      JU    BYT0;	//-> 0 Bytes (keine)
      JU    BYT1;	//-> 1 Bytes (byte)
      JU    BYT2;	//-> 2 Bytes (word)
      JU    BYT0;	//-> 3 Bytes 
      JU    BYT4;	//-> 4 Bytes (dword)
BYT0: L     DW#16#0;	//ungueltig bzw. 0/3 Fehlerbytes
      JU    KLGO;
BYT1: L     DIB [AR1,P#0.0];	//1 Fehlerbytes
      SLD   24;	//ausrichten
      JU    KLGO;
BYT2: L     DIW [AR1,P#0.0];	//2 Fehlerbytes
      SLD   16;	//ausrichten
      JU    KLGO;
BYT4: L     DID [AR1,P#0.0];	//4 Fehlerbytes
KLGO: T     DID [AR2,P#12.0];	//in akt. Fach eintragen
      CAD;	//Tausche Akku-Inhalte (LL,LH,HL,HH)
      T     #TEMP_VAR_1;	//-> sichern
//Ermittlung der Bits in der Fehlerinfo -> Bildung eindeutiger Error-Code
      L     0;	//Bit_Zaehler initialisieren
      T     #TEMP_VAR_2;
      L     32;	//Anzahl der Bits im Dword
NXB4: T     #LOOP_CNT_1;	//-> Schleifenzaehler
      L     #TEMP_VAR_2;
      INC   1;	//Bit_Zaehler erhoehen
      T     #TEMP_VAR_2;
      L     #TEMP_VAR_1;	//Unterstes Bit rausschieben
      SRD   1;
      T     #TEMP_VAR_1;	//Wenn Fehlerbit gesetzt
      JN    ERRB;	//-> Error_Code generieren
      L     #LOOP_CNT_1;
      LOOP  NXB4;
ERRB: L     #ERROR_TYPE;	//Kanaltyp ausmaskieren
      AW    W#16#F;
      SLW   5;	//* 32 (da 32 Fehlerbits pro Kanaltyp)
      +     32;	//+ 32 (Offset)
      L     #TEMP_VAR_2;	//+ Bit_Zaehler
      +I;	//= Error_Code
      T     DIW [AR2,P#20.0];	//in akt. Fach eintragen 
      L     DIB 49;	//Fehlernummer inkrementieren
      INC   1;
      T     DIB 49;
      T     DIB [AR2,P#4.0];	//und in akt. Fach eintragen
      L     DIB 48;	//Bis vorletzter Eintrag
      L     0;
      >I;
      JC    OUT;	//-> sofort Datenausgabe
      L     P##DIAG_DAT_NORM;	//Startadresse Diagnosefach
      L     DIB 45;	//+ aktuelle Gesamtdiagnoselaenge
      SLD   3;
      +D;
      T     DID 38;	//-> neuer Error_Tippindex
      L     P##DIAG_DAT_NORM;	//Gesamtlaenge der Diagnose 
      L     DIB 44;
      SLD   3;
      +D;
      L     DID 38;	//> Error_Tippindex
      >D;
      JC    OUT;	//-> Datenausgabe 
      JU    DEND;	//sonst Diagnoseende erreicht
//Wenn kein Modulstatus oder Diagnosealarm (DS0/1) vorliegt, erfolgt 
//keine detaillierte Auswertung -> herstellerspezifische Geraetediagnose.
//Handelt es sich bei dem S7-Diagnosealarm um einen gehenden Alarm bzw.   
//sind in den S7-Alarminfos (DS0/1) keine Infos enthalten, so wird eine 
//anfaenglich uebersprungene Kennungsdiagnose anschliessend ausgewertet.
KAUS: L     DW#16#0;	//Initialisieren: Steckplatznummer,
      T     DID [AR2,P#8.0];	//Modulstatus, Kanalnummer, Kanaltyp
      T     DID [AR2,P#12.0];	//Kanal-Fehlerinfos_1
      T     DID [AR2,P#16.0];	//Kanal-Fehlerinfos_2
      T     DIW [AR2,P#20.0];	//Error-Code
      T     DIW [AR2,P#4.0];	//Error-Nr. und Error-Typ
      A     DIX 31.3;	//Wenn keine Diagnoseinfos vorliegen
      JC    NODG;	//-> allg. Geraetediagnose ausgeben
      A     DIX 31.1;	//Wenn S7-Diagnosealarm (gehend)
      A     DIX 30.7;	//und Kennungsdiagnose vorhanden
      JC    BEND;	//-> Kennungsdiagnose auswerten
      AN    DIX [AR2,P#1.0];	//Wenn Slave nicht ausgefallen
      AN    DIX [AR2,P#1.1];	//und Slave nicht gestoert
      O     DIX 31.1;	//oder S7-Diagnosealarm
      JC    NGER;	//-> keine Geraetediagnose eintragen
NODG: L     B#16#5;	//sonst Error_Typ =5 (Geraetediagnose) 
      T     #SUM_SLAVES_DIAG;	//in akt. Fach eintragen
      L     545;	//Error_Code =545
      T     DIW [AR2,P#20.0];	//in akt. Fach eintragen
//DS0 oder falscher Kanaltyp im DS1 bzw. kein Kanalfehler vorhanden
//oder allgemeine Geraetediagnose ohne Detailinfos
NCHL: L     DIB 49;	//Fehlernummer erhoehen
      INC   1;
      T     DIB 49;
      T     DIB [AR2,P#4.0];	//und in akt. Fach eintragen
NGER: L     DID 38;	//Error_Tippindex inkrementieren
      L     DIB 46;	//um die Laenge des Diagnoseblocks
      SLD   3;
      +D;
      T     DID 38;
      L     P##DIAG_DAT_NORM;	//Gesamtlaenge der Diagnose 
      L     DIB 44;
      SLD   3;
      +D;
      L     DID 38;	//> Error_Tippindex
      >D;
      JC    OUT;	//-> Datenausgabe 
      JU    DEND;	//sonst Diagnoseende erreicht
//Beginn Auswertung Modulstatus
MLGO: A     DIX 30.1;	//Wenn erstmalige Blockauswertung
      JC    MODL;
      S     DIX 30.1;	//-> Start Diagnoseblock setzen
      L     DIB 46;	//Laenge des akt. Diagnoseblocks
      DEC   4;	//- 4 Byte Headerlaenge
      SLW   2;	//* 4 Module pro Byte (2 Bits pro Modul)
      T     DIB 48;	//-> Indexzaehler im Diagnoseblock
      L     DID 38;	//Error_Tippindex um Kopfbytes erhoehen
      L     P#4.0;
      +D;
      T     DID 38;
      L     DW#16#0;	//Initialisieren: Modulnummer,
      T     DID [AR2,P#8.0];	//Modulstatus, Kanalnummer, Kanaltyp
      T     DID [AR2,P#12.0];	//Kanal-Fehlerinfos_1 
      T     DID [AR2,P#16.0];	//Kanal-Fehlerinfos_2 
      T     DIW [AR2,P#20.0];	//Error-Code
MODL: L     DIB 48;	//Indexzaehler im Diagnoseblock
LPMD: T     #LOOP_CNT_1;	//-> Schleifenzaehler
      LAR1  DID 38;
      L     DIB [AR2,P#8.0];	//Modulnummer inkrementieren 
      INC   1;	//und in akt. Fach eintragen
      T     DIB [AR2,P#8.0];
      L     DIB 48;	//Indexzaehler dekrementieren
      DEC   1;
      T     DIB 48;
      L     DID 38;	//Error_Tippindex inkrementieren
      L     P#0.2;
      +D;
      T     DID 38;
      A     DIX [AR1,P#0.0];	//Wenn Statusbits <>0
      O     DIX [AR1,P#0.1];
      JC    GFMD;	//-> Fehlerauswertung
      L     #LOOP_CNT_1;
      LOOP  LPMD;	//Wenn kein Fehler gefunden
      JU    BEND;	//-> Ende Diagnoseblock
//Fehler wird gefunden im Modulstatus
GFMD: A     DIX [AR1,P#0.0];	//Modulstatus
      =     DIX [AR2,P#9.0];	//in akt. Fach eintragen
      A     DIX [AR1,P#0.1];
      =     DIX [AR2,P#9.1];
      L     B#16#2;	//Error_Typ =2 
      T     #SUM_SLAVES_DIAG;	//in akt. Fach eintragen
      L     DIB 49;	//Fehlernummer inkrementieren
      INC   1;
      T     DIB 49;
      T     DIB [AR2,P#4.0];	//und in akt. Fach eintragen
      L     DIB 48;	//Bis vorletzter Eintrag
      L     0;
      >I;
      JC    OUT;	//-> sofort Datenausgabe
      L     P##DIAG_DAT_NORM;	//Startadresse Diagnosefach
      L     DIB 45;	//+ aktuelle Gesamtdiagnoselaenge
      SLD   3;
      +D;
      T     DID 38;	//-> neuer Error_Tippindex
      L     P##DIAG_DAT_NORM;	//Gesamtlaenge der Diagnose 
      L     DIB 44;
      SLD   3;
      +D;
      L     DID 38;	//> Error_Tippindex
      >D;
      JC    OUT;	//-> Datenausgabe 
      JU    DEND;	//sonst Diagnoseende erreicht
//Beginn Auswertung Kennungsbezogene Diagnose
//Sind neben Kennungsdiagnose noch weitere Diagnosebloecke vorhanden,
//dann wird die Kennungsdiagnose nicht ausgewertet (zu wenig Infogehalt).
//Ist aber bei S7-Slaves die Geraetediagnose ohne Infos, erfolgt nach 
//anfaenglichem Ueberspringen eine neue Auswertung der Kennungsdiagnose. 
KENB: LAR2  P##ACT_DAT;	//Startadresse aktuelles Fach
      A     DIX 30.1;	//Wenn erstmalige Blockauswertung
      JC    KNGO;
      S     DIX 30.1;	//-> Start Diagnoseblock setzen
      L     DIB 46;	//Laenge des akt. Diagnoseblocks
      DEC   1;	//- 1 Byte Headerlaenge
      SLW   3;	//* 8 Bits pro Byte
      T     DIB 48;	//-> Indexzaehler im Diagnoseblock
      L     DID 38;	//Error_Tippindex um Kopfbyte erhoehen
      L     P#1.0;
      +D;
      T     DID 38;
      L     DW#16#0;	//Initialisieren: Kennungsnummer,
      T     DID [AR2,P#8.0];	//Modulstatus, Kanalnummer, Kanaltyp
      T     DID [AR2,P#12.0];	//Kanal-Fehlerinfos_1 
      T     DID [AR2,P#16.0];	//Kanal-Fehlerinfos_2 
      T     DIW [AR2,P#20.0];	//Error-Code
KNGO: L     DIB 48;	//Indexzaehler im Diagnoseblock
LPKN: T     #LOOP_CNT_1;	//-> Schleifenzaehler
      LAR1  DID 38;
      L     DIB [AR2,P#8.0];	//Kennungsnummer inkrementieren 
      INC   1;	//und in akt. Fach eintragen
      T     DIB [AR2,P#8.0];
      L     DIB 48;	//Indexzaehler dekrementieren
      DEC   1;
      T     DIB 48;
      L     DID 38;	//Error_Tippindex inkrementieren
      L     P#0.1;
      +D;
      T     DID 38;
      A     DIX [AR1,P#0.0];	//Wenn Kennung gesetzt
      JC    GFKN;	//-> Fehlerauswertung
      L     #LOOP_CNT_1;
      LOOP  LPKN;	//Wenn kein Fehler gefunden
      JU    BEND;	//-> Ende Diagnoseblock
//Fehler wird gefunden in der Kennungsdiagnose
GFKN: A     DIX 30.7;	//Wenn Kennungsdiagnose vorhanden
      AN    DIX 31.0;	//und bisher keine Kanaldiagnose 
      AN    DIX 31.2;	//und bisher keine S7-Diagnose 
      JC    KEGO;	//-> neue bzw. weitere Auswertung
      S     DIX 30.7;	//sonst Erst-Erkennung setzen
      L     DIB 44;	//Wenn SFC13-Diagnoselaenge
      L     DIB 45;	//> aktuelle Gesamtdiagnoselaenge
      >I;
      JC    BEND;	//-> Keine Kennungsdiagnose auswerten
KEGO: L     B#16#1;	//Error_Typ =1 
      T     #SUM_SLAVES_DIAG;	//in akt. Fach eintragen
      L     DIB 49;	//Fehlernummer inkrementieren
      INC   1;
      T     DIB 49;
      T     DIB [AR2,P#4.0];	//und in akt. Fach eintragen
      L     DIB 48;	//Bis vorletzter Eintrag
      L     0;
      >I;
      JC    OUT;	//-> sofort Datenausgabe
      L     P##DIAG_DAT_NORM;	//Startadresse Diagnosefach
      L     DIB 45;	//+ aktuelle Gesamtdiagnoselaenge
      SLD   3;
      +D;
      T     DID 38;	//-> neuer Error_Tippindex
      L     P##DIAG_DAT_NORM;	//Gesamtlaenge der Diagnose 
      L     DIB 44;
      SLD   3;
      +D;
      L     DID 38;	//> Error_Tippindex
      >D;
      JC    OUT;	//-> Datenausgabe 
      JU    DEND;	//sonst Diagnoseende erreicht
//Beginn Auswertung Kanalbezogene Diagnose (immer 3 Bytes lang)
KANB: S     DIX 31.0;	//Kanaldiagnose vorhanden
      R     DIX 30.0;	//Error_TIPP-Start ruecksetzen
      LAR2  P##ACT_DAT;	//Startadresse aktuelles Fach
      L     DW#16#0;	//Initialisieren: Kennungsnummer,
      T     DID [AR2,P#8.0];	//Modulstatus, Kanalnummer, Kanaltyp
      T     DID [AR2,P#12.0];	//Kanal-Fehlerinfos_1 
      T     DID [AR2,P#16.0];	//Kanal-Fehlerinfos_2 
      T     DIW [AR2,P#20.0];	//Error-Code
      LAR1  DID 38;	//Error_Tippindex
      L     DIB [AR1,P#0.0];	//Header(Bit7,6:HeaderCode/5-0:KennungsNr)
      AW    W#16#3F;	//Kanalkennungsnummer ermitteln
      INC   1;
      T     DIB [AR2,P#8.0];	//in akt. Fach eintragen
      L     DIB [AR1,P#1.0];	//Kanalnummer ermitteln
      AW    W#16#3F;
      T     #ERROR_NO;	//in akt. Fach eintragen
      L     DIB [AR1,P#1.0];	//Kanaltyp (nach Norm) ermitteln
      SRW   6;	//00=Res, 01=In, 02=Out, 03=In/Out
      T     #ERROR_TYPE;	//in akt. Fach eintragen
//Fehlerinfo bilden, indem der ermittelte Error_Code ueber "2^Error_Code"
//bitcodiert wird.
      L     DW#16#1;	//Fehlerinfo vorbelegen
      T     #TEMP_VAR_1;
      L     B#16#0;
      L     DIB [AR1,P#2.0];	//Fehlertyp
      AW    W#16#1F;	//ausmaskieren -> Error_Code
      T     DIW [AR2,P#20.0];	//in akt. Fach eintragen
      ==I;	//Wenn Error_Code =0
      JC    NCOD;	//-> keine weitere Fehlerinfo-Kodierung 
ZEXP: T     #LOOP_CNT_1;	//Schleifenzaehler =Error_Code
      L     #TEMP_VAR_1;	//Fehlerinfo * 2 (potenzieren)
      SLD   1;
      T     #TEMP_VAR_1;
      L     #LOOP_CNT_1;
      LOOP  ZEXP;
NCOD: L     #TEMP_VAR_1;	//Bitcodierte Fehlerinfo
      CAD;	//Tausche Akku-Inhalte (LL,LH,HL,HH)   
      T     DID [AR2,P#12.0];	//in akt. Fach eintragen
      L     B#16#3;	//Error_Typ =3 
      T     #SUM_SLAVES_DIAG;	//in akt. Fach eintragen
      L     DIB 49;	//Fehlernummer inkrementieren
      INC   1;
      T     DIB 49;
      T     DIB [AR2,P#4.0];	//und in akt. Fach eintragen
      L     DID 38;	//Error_Tippindex inkrementieren
      L     P#3.0;	//um die Laenge des Diagnoseblocks
      +D;
      T     DID 38;
      L     P##DIAG_DAT_NORM;	//Gesamtlaenge der Diagnose 
      L     DIB 44;
      SLD   3;
      +D;
      L     DID 38;	//> Error_Tippindex
      >D;
      JC    OUT;	//-> Datenausgabe 
//An diese Stelle kommt das Programm nur, wenn bei der Fehlersuche im 
//Diagnoseblock ein Fehler gefunden wurde und der Error-Tippindex das 
//Ende des Diagnosetelegramms erreicht hat. Dann wird beim naechsten
//Fehler-Tippen wieder beim ersten Diagnoseblock des Diagnosetelegramms
//begonnen.
DEND: R     DIX 30.0;	//Error_TIPP-Start ruecksetzen
      L     DIB 49;	//Fehlernummer
      T     DIB [AR2,P#4.0];	//in akt. Fach eintragen
      L     6;	//Akt. Diaglaenge initialisieren
      T     DIB 45;	//mit 6 Bytes Normdiagnose
      L     0;	//Initialisieren
      T     DIB 46;	//Initialsieren Blocklaenge
      T     DIB 49;	//Fehlernummer =0 setzen
      L     P##DIAG_DAT_NORM;
      T     DID 38;	//Error_Tippindex 
      JU    OUT;	//-> Datenausgabe
//An diese Stelle kommt das Programm nur, wenn bei der Fehlersuche im 
//Diagnoseblock kein Fehler gefunden wurde. Dann wird geprueft, ob das
//Blockende auch gleichzeitig das Ende des gesamten Diagnosetelegramms
//bedeutet. Wenn ja, faengt die Fehlerauswertung sofort beim ersten 
//Diagnoseblock des Diagnosetelegramms wieder an. Ansonsten wird beim 
//naechst folgenden Diagnoseblock weiter nach Fehlern gesucht.
BEND: L     DIB 44;	//Wenn SFC13-Diagnoselaenge 
      L     DIB 45;	//> Aktuelle Gesamtdiagnoselaenge
      >I;
      JC    NBLK;	//-> naechsten Diagblock auswerten
      L     6;	//Akt. Diaglaenge initialisieren
      T     DIB 45;	//mit 6 Bytes Normdiagnose
      L     0;
      T     DIB 46;	//Initialisieren Blocklaenge
      T     DIB 49;	//Fehlernummer =0 setzen
      T     DIB 48;	//Indexzaehler im Diagblock loeschen
      T     DIB [AR2,P#8.0];	//Kennungs- bzw. Modul-Nr. loeschen 
      L     P##DIAG_DAT_NORM;
      T     DID 38;	//Error_Tippindex =Start Diagnose
      A(;
      L     DIB [AR2,P#4.0];	//Wenn bisher keine Fehler gefunden
      L     0;
      ==I;
      );
      AN    DIX 30.7;	//und keine Kenn.diagnose vorhanden
      R     DIX 30.0;	//-> Error_TIPP-Start ruecksetzen
      JC    OUT;	//-> weiter Datenausgabe
      JU    NBLK;	//sonst ersten Diagblock auswerten
NETWORK
TITLE = Versorgung der Ausgangsparameter
//Die Daten aus dem aktuellen Fach und die Anzahl der betroffenen Slaves werden 
//an die FB-Ausgangsparameter uebergeben. Zusaetzlich wird auf den Diagnose- 
//Zaehler des aktuell angezeigten Slaves zugegriffen und am Ausgangsparameter 
//angezeigt. 
OUT:  LAR2  P##ACT_DAT;	//Startadresse aktuelles Fach
      L     B#16#0;	//Wenn Slave_Nr. =0
      T     DIB 26;	//-> Diagnose_Zaehler vorab loeschen
      L     DIB [AR2,P#0.0];	//-> kein Diagnose_Zaehler auswerten 
      T     DIB 6;	//Slave_Nr. ausgeben
      ==I;
      JC    STAT;
      DEC   1;	//Slaveposition = Slave_Nr.-1
      SLD   3;	//Byteadresse
      L     P##DIAG_CNT;	//+ Startadresse Diagnose_Zaehler
      +D;
      LAR1;
      L     DIB [AR1,P#0.0];	//Diag_Zaehler des Slaves lesen
      T     DIB 26;	//und ausgeben
STAT: L     DIB [AR2,P#1.0];
      T     DIB 7;	//Slave_Status ausgeben
      L     DIW [AR2,P#2.0];
      T     DIW 8;	//Ident_Number (PNO-ID) ausgeben
      L     DIB [AR2,P#4.0];
      T     DIB 10;	//Error_Nr. ausgeben
      L     #SUM_SLAVES_DIAG;
      T     DIB 11;	//Error_Typ ausgeben
//In Fach 6 und 7 liegt die Diagnoseadresse des Slaves.
      L     DIB [AR2,P#8.0];
      T     DIB 12;	//Modul_Nr. ausgeben
      L     DIB [AR2,P#9.0];
      T     DIB 13;	//Modul_Status ausgeben
      L     #ERROR_NO;
      T     DIB 14;	//Kanal_Nr. ausgeben
      L     #ERROR_TYPE;
      T     DIB 15;	//Kanal_Typ ausgeben
      L     DIW [AR2,P#20.0];
      T     DIW 16;	//Kanal_Errorcode
      L     DID [AR2,P#12.0];
      T     DID 18;	//Kanal_Fehlerinfos_1 ausgeben
      L     DID [AR2,P#16.0];
      T     DID 22;	//Kanal_Fehlerinfos_2 ausgeben
      L     DIB 32;
      T     DIB 5;	//Summe der Betr_Slaves ausgeben
NETWORK
TITLE = OK-Bit, BUSY-Bit, Tippindex, Interrupts freigeben
//Sind keine Slaves betroffen (ausgefallen oder gestoert), wird das O.K.-Bit 
//gesetzt und der Slave- und Error-Tippindex initialisiert. Bei falscher 
//Bausteinparametrierung wird der Inhalt des Eingangsparameters Mastersystem-ID 
//in das C91-Fach eingetragen. Ist RESET aktiviert, wird die Init-Routine 
//bearbeitet. Abschliessend werden die Interrupts wieder freigegeben. 
ENDE: L     DIB 32;	//Wenn Anzahl Betr_Slaves =0
      L     0;
      ==I;
      JCN   BUSY;
      S     DIX 4.0;	//-> Alles_O.K.-Bit setzen
      R     DIX 29.7;	//-> Tippstart Slaves ruecksetzen
      R     DIX 30.0;	//-> Tippstart Fehler ruecksetzen
      L     P##AFFECT_SLAVES;	//-> Slave_Tippindex initialisieren
      T     DID 34;
      L     P##DIAG_DAT_NORM;	//-> Error_Tippindex initialisieren
      T     DID 38;
      L     1;	//-> Slaveadresse initialisieren
      T     DIW 50;
BUSY: A     DIX 1402.4;	//Wenn Reset aktiviert
      FP    DIX 29.5;
      S     DIX 30.3;	//sichern
      A     DIX 30.4;	//Wenn Parametrierfehler
      O(;	//oder
      A     DIX 28.4;	//Wenn Anlauf/Resetroutine beendet
      AN    DIX 28.7;	//     und kein SFC13-Lesen aktiv
      AN    DIX 29.0;	//     und kein SZLC91-Lesen aktiv
      A(;	//     und 
      AN    DIX 29.2;	//         kein Folgeauftrag vorh.
      O(;	//         oder
      A     DIX 29.2;	//         Folgeauftrag vorh.
      A     DIX 30.3;	//         aber Reset aktiviert  
      );
      );
      );
      R     DIX 27.1;	//-> FB-Bearbeitung beendet
      AN    DIX 30.4;	//Wenn Parametrierfehler
      JC    PROK;
      LAR1  P##SZL_READ_C91;	//Startadresse C91-Fach (BGZD)
      L     #MAST_SYSTEM_ID;	//Eingangsparameter Mastersystem-ID 
      T     DIB [AR1,P#0.0];	//in C91-Fach eintragen
PROK: AN    DIX 27.1;	//Wenn BUSY =0
      A     DIX 30.3;	//und Reset aktiv
      JC    RSET;	//-> alles initialisieren
      A     DIX 30.6;	//BIE-Bit sichern
      SAVE;
      CALL  "EN_AIRT" (
           RET_VAL                  := #RETVAL_SFC);	//Verz. Interrupts wieder freigeben
END_FUNCTION_BLOCK

// FB 523: know-how protected block, not included

// FB 913: know-how protected block, not included

// FB 914: know-how protected block, not included

// FB 915: know-how protected block, not included

FUNCTION_BLOCK "Job_List"	// FB 919
TITLE = Job_List
//V1.1
AUTHOR : SIEMENS
FAMILY : COMM
NAME : JOB_LIST
VERSION : 1.1
VAR_INPUT
  CYCLICAL : TIME ;	//Cyclical time to start the job list
  DONE : BOOL ;	//Job finished without error (from MODBUS block)
  ERROR : BOOL ;	//Job finished with error (from MODBUS block)
  Job1_DATA_TYPE : BYTE ;	//1st job: data type (1-4)
  Job1_START_ADDRESS : WORD ;	//Start address (register or bit)
  Job1_LENGTH : WORD ;	//Count of registers/bits
  Job1_WRITE_READ : BOOL ;	//TRUE = write, FALSE = read
  Job2_DATA_TYPE : BYTE ;	//2nd job: data type (1-4)
  Job2_START_ADDRESS : WORD ;	//Start address (register or bit)
  Job2_LENGTH : WORD ;	//Count of registers/bits
  Job2_WRITE_READ : BOOL ;	//TRUE = write, FALSE = read
  Job3_DATA_TYPE : BYTE ;	//3rd job: data type (1-4)
  Job3_START_ADDRESS : WORD ;	//Start address (register or bit)
  Job3_LENGTH : WORD ;	//Count of registers/bits
  Job3_WRITE_READ : BOOL ;	//TRUE = write, FALSE = read
  Job4_DATA_TYPE : BYTE ;	//4th job: data type (1-4)
  Job4_START_ADDRESS : WORD ;	//Start address (register or bit)
  Job4_LENGTH : WORD ;	//Count of registers/bits
  Job4_WRITE_READ : BOOL ;	//TRUE = write, FALSE = read
  Job5_DATA_TYPE : BYTE ;	//5th job: data type (1-4)
  Job5_START_ADDRESS : WORD ;	//Start address (register or bit)
  Job5_LENGTH : WORD ;	//Count of registers/bits
  Job5_WRITE_READ : BOOL ;	//TRUE = write, FALSE = read
  Job6_DATA_TYPE : BYTE ;	//1st job: data type (1-4)
  Job6_START_ADDRESS : WORD ;	//Start address (register or bit)
  Job6_LENGTH : WORD ;	//Count of registers/bits
  Job6_WRITE_READ : BOOL ;	//TRUE = write, FALSE = read
  Job7_DATA_TYPE : BYTE ;	//2nd job: data type (1-4)
  Job7_START_ADDRESS : WORD ;	//Start address (register or bit)
  Job7_LENGTH : WORD ;	//Count of registers/bits
  Job7_WRITE_READ : BOOL ;	//TRUE = write, FALSE = read
  Job8_DATA_TYPE : BYTE ;	//3rd job: data type (1-4)
  Job8_START_ADDRESS : WORD ;	//Start address (register or bit)
  Job8_LENGTH : WORD ;	//Count of registers/bits
  Job8_WRITE_READ : BOOL ;	//TRUE = write, FALSE = read
  Job9_DATA_TYPE : BYTE ;	//4th job: data type (1-4)
  Job9_START_ADDRESS : WORD ;	//Start address (register or bit)
  Job9_LENGTH : WORD ;	//Count of registers/bits
  Job9_WRITE_READ : BOOL ;	//TRUE = write, FALSE = read
  Job10_DATA_TYPE : BYTE ;	//5th job: data type (1-4)
  Job10_START_ADDRESS : WORD ;	//Start address (register or bit)
  Job10_LENGTH : WORD ;	//Count of registers/bits
  Job10_WRITE_READ : BOOL ;	//TRUE = write, FALSE = read
END_VAR
VAR_OUTPUT
  QENQ : BOOL ;	//Job initiation
  QDATA_TYPE : BYTE ;	//Data type 1:Coils, 2:Inputs, 3:Holding, 4:Input Registers
  QSTART_ADDRESS : WORD ;	//Start address (register or bit)
  QLENGTH : WORD ;	//Count of registers/bits
  QWRITE_READ : BOOL ;	//TRUE = write, FALSE = read
  BUSY : BOOL ;	//Job list processing
  STATUS : WORD ;	//Status information of job list block
END_VAR
VAR_IN_OUT
  ABORT : BOOL ;	//Reset: Stop the processing of the job list
END_VAR
VAR
  Count_of_Jobs : INT  := 10;	//Count of Jobs in the input area
  TON_JOB : SFB 4;	//Timer for cyclical processing
  Current_Job : INT ;	//Current processed job
  i : INT ;	//internal counter
  sIDB_Nr : WORD ;	//number of instance data block
  Next_Job : BOOL ;	//TRUE: next job should be start
  Wait : BOOL ;	//internal use
END_VAR
VAR_TEMP
  address_Struct : STRUCT
   ANY_id : WORD ;
   Length : WORD ;
   DB_Number : WORD ;
   Byte_Pointer : DWORD ;
  END_STRUCT ;
END_VAR
BEGIN
// body was compiled from an SCL source; compiled code not shown
END_FUNCTION_BLOCK

FUNCTION_BLOCK "JOB_RESET"	// FB 921
VERSION : 0.0
VAR_INPUT
  CMD : BOOL ;
  SOURSE_DB : BLOCK_DB ;
  TARGET_DB : BLOCK_DB ;
END_VAR
VAR
  I : INT ;	//Static Variables
END_VAR
BEGIN
// body was compiled from an SCL source; compiled code not shown
END_FUNCTION_BLOCK

// FB 1071: know-how protected block, not included

// FB 1501: know-how protected block, not included

FUNCTION_BLOCK "HF3_PID_FB2005"	// FB 2005
TITLE = PID
VERSION : 0.1
VAR_INPUT
  COM_RST : BOOL ;
  MAN_ON { S7_m_c := 'true' }: BOOL  := TRUE;	//1-手动，0-自动
  PVPER_ON : BOOL ;	//0-设定的过程变量；1-来自IO的过程变量
  P_SEL : BOOL  := TRUE;	//P 选择开关
  I_SEL : BOOL  := TRUE;	//I 选择开关
  INT_HOLD : BOOL ;	//INTEGRAL ACTION HOLD 积分器被冻结
  I_ITL_ON : BOOL ;	//INITIALIZATION OF THE INTEGRAL 积分器初始值
  D_SEL : BOOL ;	//DERIVATIVE ACTION ON可以单独激活或失去D作用
  INT_EXT { S7_m_c := 'true' }: BOOL ;	//0＝内部设定，1＝外部设定
  IN_1 : BOOL ;	//Spare
  IN_2 : BOOL ;	//Spare
  IN_3 : BOOL ;	//Backup
  PV_PER : WORD ;	//PROCESS VARIABLE PERIPHERAL
  SP_INT { S7_m_c := 'true'; S7_archive := 'shortterm' }: REAL ;	//PID内部设定值
  UNIT { S7_m_c := 'true' }: INT ;	//Unit
  PV_IN { S7_m_c := 'true'; S7_archive := 'shortterm' }: REAL ;	//实际输入值
  GAIN { S7_m_c := 'true' }: REAL  := 2.000000e+000;	//比例
  TI { S7_m_c := 'true' }: DINT  := L#10;	//积分时间
  TD { S7_m_c := 'true' }: DINT  := L#10;	//微分时间
  CYCLE : TIME  := T#1S;
  TM_LAG : TIME  := T#2S;	//TIME LAG OF THE DERIVATIVE ACTION微分延时时间
  DEADB_W { S7_m_c := 'true' }: REAL ;	//死区
  LMN_HLM { S7_m_c := 'true' }: REAL  := 1.000000e+002;	//输出上限
  LMN_LLM { S7_m_c := 'true' }: REAL ;	//输出下限
  PV_FAC : REAL  := 1.000000e+000;	//实际输入因子  （通常为"1"）
  PV_OFF : REAL ;	//实际输入补偿  （通常不需要）
  LMN_FAC : REAL  := 1.000000e+000;	//输出因子  （通常为"1"）
  LMN_OFF : REAL ;	//输出补偿  （通常不需要）
  I_ITLVAL : REAL ;	//积分初始值
  DISV : REAL ;	//前馈值
  SP_EXT { S7_m_c := 'true' }: REAL ;	//逻辑外部设定值（外环输出值）
  IN_4 : REAL ;	//Spare
  PV_RANG_L : REAL ;
  PV_RANG_H : REAL  := 1.000000e+002;
END_VAR
VAR_OUTPUT
  QLMN_HLM : BOOL ;	//手动值高限
  QLMN_LLM : BOOL ;	//手动值底限
  QMAN_ON { S7_m_c := 'true' }: BOOL ;	//PID手自动状态，0-手动，1-自动
  OUT_1 : BOOL ;	//Spare
  OUT_2 : BOOL ;	//Spare
  OUT_3 : BOOL ;	//Spare
  LMN_PER { S7_m_c := 'true' }: WORD ;	//预设手动值
  LMN_P { S7_m_c := 'true' }: REAL ;	//PROPORTIONAL COMPONENT
  LMN_I { S7_m_c := 'true' }: REAL ;	//INTEGRAL COMPONENT
  LMN_D { S7_m_c := 'true' }: REAL ;	//DERIVATIVE COMPONENT
  PV { S7_m_c := 'true' }: REAL ;	//过程值
  ER { S7_m_c := 'true' }: REAL ;	//错误信号
  OUT_4 : BOOL ;	//Spare
END_VAR
VAR_IN_OUT
  MAN { S7_m_c := 'true'; S7_archive := 'shortterm' }: REAL ;	//手动输出值
  LMN { S7_m_c := 'true'; S7_archive := 'shortterm' }: REAL ;	//PID输出
  IN_OUT_1 : BOOL ;
  IN_OUT_2 : BOOL ;
  IN_OUT_3 : REAL ;
  SP_M { S7_m_c := 'true' }: REAL ;	//SP实际设定值
END_VAR
VAR
  PID_CTRL : FB 41;
  TI_M : DINT ;
  TD_M : DINT ;
  TI_TIME : TIME ;
  TD_TIME : TIME ;
END_VAR
BEGIN
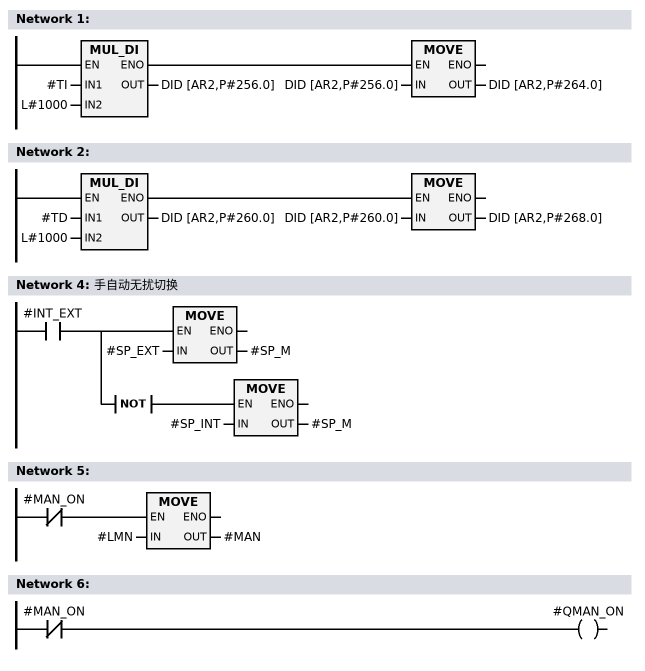
NETWORK
TITLE =
//Intergration Time
      A(;
      L     #TI;
      L     L#1000;
      *D;
      T     DID [AR2,P#256.0];
      AN    OV;
      SAVE;
      CLR;
      A     BR;
      );
      JNB   _001;
      L     DID [AR2,P#256.0];
      T     DID [AR2,P#264.0];
_001: NOP   0;
NETWORK
TITLE =
//Derivative Time
      A(;
      L     #TD;
      L     L#1000;
      *D;
      T     DID [AR2,P#260.0];
      AN    OV;
      SAVE;
      CLR;
      A     BR;
      );
      JNB   _002;
      L     DID [AR2,P#260.0];
      T     DID [AR2,P#268.0];
_002: NOP   0;
NETWORK
TITLE =
//Cont_C
      A     #COM_RST;
      =     L 0.0;
      BLD   103;
      A     #MAN_ON;
      =     L 0.1;
      BLD   103;
      A     #PVPER_ON;
      =     L 0.2;
      BLD   103;
      A     #P_SEL;
      =     L 0.3;
      BLD   103;
      A     #I_SEL;
      =     L 0.4;
      BLD   103;
      A     #INT_HOLD;
      =     L 0.5;
      BLD   103;
      A     #I_ITL_ON;
      =     L 0.6;
      BLD   103;
      A     #D_SEL;
      =     L 0.7;
      BLD   103;
      BLD   14;
      =     L 7.0;
      L     DINO;
      T     LW 5;
      CDB;
      OPN   DI [LW 5];
      TAR2  LD 1;
      A     L 0.0;
      =     DIX [AR2,P#130.0];
      A     L 0.1;
      =     DIX [AR2,P#130.1];
      A     L 0.2;
      =     DIX [AR2,P#130.2];
      A     L 0.3;
      =     DIX [AR2,P#130.3];
      A     L 0.4;
      =     DIX [AR2,P#130.4];
      A     L 0.5;
      =     DIX [AR2,P#130.5];
      A     L 0.6;
      =     DIX [AR2,P#130.6];
      A     L 0.7;
      =     DIX [AR2,P#130.7];
      L     DBD [AR2,P#26.0];
      T     DID [AR2,P#132.0];
      L     DBD [AR2,P#126.0];
      T     DID [AR2,P#136.0];
      L     DBD [AR2,P#10.0];
      T     DID [AR2,P#140.0];
      L     DBW [AR2,P#2.0];
      T     DIW [AR2,P#144.0];
      L     DBD [AR2,P#112.0];
      T     DID [AR2,P#146.0];
      L     DBD [AR2,P#14.0];
      T     DID [AR2,P#150.0];
      L     DBD [AR2,P#264.0];
      T     DID [AR2,P#154.0];
      L     DBD [AR2,P#268.0];
      T     DID [AR2,P#158.0];
      L     DBD [AR2,P#30.0];
      T     DID [AR2,P#162.0];
      L     DBD [AR2,P#34.0];
      T     DID [AR2,P#166.0];
      L     DBD [AR2,P#38.0];
      T     DID [AR2,P#170.0];
      L     DBD [AR2,P#42.0];
      T     DID [AR2,P#174.0];
      L     DBD [AR2,P#46.0];
      T     DID [AR2,P#178.0];
      L     DBD [AR2,P#50.0];
      T     DID [AR2,P#182.0];
      L     DBD [AR2,P#54.0];
      T     DID [AR2,P#186.0];
      L     DBD [AR2,P#58.0];
      T     DID [AR2,P#190.0];
      L     DBD [AR2,P#62.0];
      T     DID [AR2,P#194.0];
      L     DBD [AR2,P#66.0];
      T     DID [AR2,P#198.0];
      +AR2  P#130.0;
      UC    "pid";
      LAR2  LD 1;
      L     DID [AR2,P#202.0];
      T     DBD [AR2,P#116.0];
      L     DIW [AR2,P#206.0];
      T     DBW [AR2,P#88.0];
      A     DIX [AR2,P#208.0];
      =     DBX [AR2,P#86.0];
      A     DIX [AR2,P#208.1];
      =     DBX [AR2,P#86.1];
      L     DID [AR2,P#210.0];
      T     DBD [AR2,P#90.0];
      L     DID [AR2,P#214.0];
      T     DBD [AR2,P#94.0];
      L     DID [AR2,P#218.0];
      T     DBD [AR2,P#98.0];
      L     DID [AR2,P#222.0];
      T     DBD [AR2,P#102.0];
      L     DID [AR2,P#226.0];
      T     DBD [AR2,P#106.0];
      CDB;
      BLD   15;
      NOP   0;
NETWORK
TITLE = 手自动无扰切换
//当外部设定时，逻辑外部设定值赋值给设定值；当内部设定时，PID内部设定值赋值给设定
//值
//。
//主要用在串级调节回路
      A     #INT_EXT;
      =     L 0.0;
      A     L 0.0;
      JNB   _003;
      L     #SP_EXT;
      T     #SP_M;
_003: NOP   0;
      A     L 0.0;
      NOT;
      JNB   _004;
      L     #SP_INT;
      T     #SP_M;
_004: NOP   0;
NETWORK
TITLE =
      AN    #MAN_ON;
      JNB   _005;
      L     #LMN;
      T     #MAN;
_005: NOP   0;
NETWORK
TITLE =
      AN    #MAN_ON;
      =     #QMAN_ON;
END_FUNCTION_BLOCK

FUNCTION_BLOCK "HF3_RunFaultSum"	// FB 2006
TITLE = TIMER_MOTOR
AUTHOR : SIEMENS
FAMILY : SIEMENS
NAME : SIEMENS
VERSION : 1.0
VAR_INPUT
  RUN : BOOL ;
  ERROR : BOOL ;
  SAMPLE_T : BOOL ;	//Cycle Time of the CPU Time plus (Seconds)
  RESET_RUN : BOOL ;
  RESET_ERROR : BOOL ;
  RESET_TIME : BOOL ;
END_VAR
VAR_OUTPUT
  RUNTIME : REAL ;	//Run Timer in Hour
  RUN_COUNTER : INT ;
  ERROR_COUNTER : INT ;
END_VAR
VAR
  RUN_SECOND : REAL ;	//RUNTIME counter in Second
  OLD_SAMPLE_T : BOOL ;
  OLD_RUN : BOOL ;
  OLD_ERROR : BOOL ;
END_VAR
BEGIN
// body was compiled from an SCL source; compiled code not shown
END_FUNCTION_BLOCK

FUNCTION_BLOCK "HF3_EPS_FB2501"	// FB 2501
TITLE = EPS 主程序端
//定义参照点表
VERSION : 0.1
VAR
  EPS21 : FB 2502;
  EPS11 : FB 2502;
END_VAR
BEGIN
NETWORK
TITLE = EPS_A
// (network holds code this reader does not know; not shown)
NETWORK
TITLE =
// (network holds code this reader does not know; not shown)
END_FUNCTION_BLOCK

FUNCTION_BLOCK "HF3_EPS_FB2502"	// FB 2502
VERSION : 0.1
VAR_INPUT
  DB_Number : INT ;
END_VAR
VAR_OUTPUT
  EPS_ToHMI1 : WORD ;
  EPS_ToHMI : ARRAY  [0 .. 15 ] OF INT ;
END_VAR
VAR
  data_p : DWORD ;	//DATA POINTER
  AR2_data : DWORD ;
END_VAR
VAR_TEMP
  dbnumber : INT ;
  DIN_TEMP : WORD ;
  NO_TEMP : INT ;
  CommOK : BOOL ;	//communication status
  AR2_Temp : DWORD ;	//current multi-instance AR2 data
END_VAR
BEGIN
NETWORK
TITLE = Initialize Parameters
      L     P#2.0;
      T     #data_p;
      L     DW#16#0;
      T     #AR2_Temp;
      L     #DB_Number;
      T     #dbnumber;
      OPN   DB [#dbnumber];
      L     DINO;
      T     #DIN_TEMP;
      OPN   DI [#DIN_TEMP];
NETWORK
TITLE = Data Output
      L     #data_p;
      LAR1;
      TAR2;
//Figure out the absolute address of Instance DB variable 
      T     #AR2_Temp;
      AD    DW#16#FFFFFF;	//Close area identifier 
      L     P##EPS_ToHMI;
      +D;
      LAR2;
//  Pass PARAMETER
      L     16;
LP:   T     #NO_TEMP;
      L     DBW [AR1,P#0.0];
      T     W [AR2,P#0.0];
      +AR1  P#2.0;
      +AR2  P#2.0;
      L     #NO_TEMP;
      LOOP  LP;
      L     #AR2_Temp;	// Recovery AR2   
      LAR2;
NETWORK
TITLE = Communication Status
      L     DBW 0;
      L     0;
      ==I;
      =     #CommOK;
NETWORK
TITLE = Pass EPS Status to HMI
      CALL  "HF3_B_T_W_FC51" (
           Bit_0                    := DBX 35.0,
           Bit_1                    := DBX 35.1,
           Bit_2                    := DBX 35.2,
           Bit_3                    := DBX 35.3,
           Bit_4                    := DBX 35.4,
           Bit_5                    := DBX 35.5,
           Bit_6                    := DBX 35.6,
           Bit_7                    := DBX 35.7,
           Bit_8                    := DBX 34.0,
           Bit_9                    := DBX 34.1,
           Bit_10                   := DBX 34.2,
           Bit_11                   := DBX 34.3,
           Bit_12                   := DBX 34.4,
           Bit_13                   := DBX 34.5,
           Bit_14                   := DBX 34.6,
           Bit_15                   := #CommOK,
           Word1                    := #EPS_ToHMI1);	//市电状态(报警点) / 逆变状态(报警点) / 综合故障(报警点) / 过载(报警点) / 强制运行(报警点) / 电池状态(报警点) / 充电状态(报警点) / 支路故障(报警点) / 电池欠压 / 市电/逆变状态 / 均/浮充 / 双切位置 / ͨѶ״̬
NETWORK
TITLE = END function block
      SET;
      SAVE;
      CLR;
      BEU;
END_FUNCTION_BLOCK

FUNCTION_BLOCK "HF3_IMCC_CommOK_FB2512"	// FB 2512
VERSION : 0.1
VAR
  CommOK : FB 2513;
END_VAR
BEGIN
NETWORK
TITLE =
      BLD   14;
      =     L 6.0;
      L     DINO;
      T     LW 4;
      CDB;
      OPN   DI [LW 4];
      TAR2  LD 0;
      OPN   DI 2291;
      L     DIW 0;
      OPN   DI [LW 4];
      T     #CommOK.inRD_IMCC_HB;
      +AR2  P#0.0;
      UC    "HF3_IMCC_CommOK_FB2513";
      LAR2  LD 0;
      A     #CommOK.IMCC_CommOK;
      =     "IMCC_Comok";
      CDB;
      BLD   15;
      NOP   0;
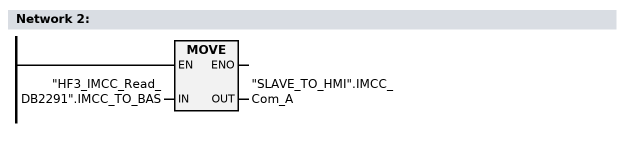
NETWORK
TITLE =
      L     "HF3_IMCC_Read_DB2291".IMCC_TO_BAS;
      T     "SLAVE_TO_HMI".IMCC_Com_A;
      NOP   0;
END_FUNCTION_BLOCK

FUNCTION_BLOCK "HF3_IMCC_CommOK_FB2513"	// FB 2513
VERSION : 0.1
VAR_INPUT
  inRD_IMCC_HB : WORD ;
END_VAR
VAR_OUTPUT
  IMCC_CommOK : BOOL ;
END_VAR
VAR
  Ton1 : SFB 4;
  CommOK1 : BOOL ;
  CommOK2 : BOOL ;
  fault1 : BOOL ;
  Ton2 : SFB 4;
  fault2 : BOOL ;
  TON3 : SFB 4;
END_VAR
BEGIN
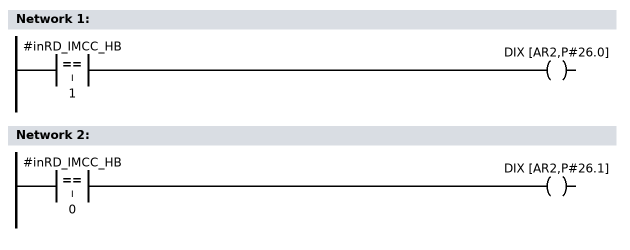
NETWORK
TITLE =
      L     #inRD_IMCC_HB;
      L     1;
      ==I;
      =     DIX [AR2,P#26.0];
NETWORK
TITLE =
      L     #inRD_IMCC_HB;
      L     0;
      ==I;
      =     DIX [AR2,P#26.1];
NETWORK
TITLE =
      A     DIX [AR2,P#26.0];
      =     L 0.0;
      BLD   103;
      BLD   16;
      =     L 7.0;
      L     DINO;
      T     LW 5;
      CDB;
      OPN   DI [LW 5];
      TAR2  LD 1;
      A     L 0.0;
      =     DIX [AR2,P#4.0];
      L     L#30000;
      T     DID [AR2,P#6.0];
      +AR2  P#4.0;
      UC    "TON";
      LAR2  LD 1;
      A     DIX [AR2,P#10.0];
      =     DBX [AR2,P#26.2];
      CDB;
      BLD   17;
      NOP   0;
NETWORK
TITLE =
      A     DIX [AR2,P#26.1];
      =     L 0.0;
      BLD   103;
      BLD   16;
      =     L 7.0;
      L     DINO;
      T     LW 5;
      CDB;
      OPN   DI [LW 5];
      TAR2  LD 1;
      A     L 0.0;
      =     DIX [AR2,P#28.0];
      L     L#30000;
      T     DID [AR2,P#30.0];
      +AR2  P#28.0;
      UC    "TON";
      LAR2  LD 1;
      A     DIX [AR2,P#34.0];
      =     DBX [AR2,P#50.0];
      CDB;
      BLD   17;
      NOP   0;
NETWORK
TITLE =
      AN    DIX [AR2,P#50.0];
      AN    DIX [AR2,P#26.2];
      =     L 0.0;
      BLD   103;
      BLD   16;
      =     L 7.0;
      L     DINO;
      T     LW 5;
      CDB;
      OPN   DI [LW 5];
      TAR2  LD 1;
      A     L 0.0;
      =     DIX [AR2,P#52.0];
      L     L#30000;
      T     DID [AR2,P#54.0];
      +AR2  P#52.0;
      UC    "TON";
      LAR2  LD 1;
      A     DIX [AR2,P#58.0];
      =     DBX [AR2,P#2.0];
      CDB;
      BLD   17;
      NOP   0;
END_FUNCTION_BLOCK

FUNCTION_BLOCK "HF3_LSQK_FB2521"	// FB 2521
VERSION : 0.1
VAR
  PT : TIME  := T#40MS;
  LSQK : FB 2522;
END_VAR
BEGIN
NETWORK
TITLE =
      BLD   14;
      =     L 7.0;
      L     DINO;
      T     LW 5;
      CDB;
      OPN   DI [LW 5];
      TAR2  LD 1;
      OPN   DI 6001;
      L     DIW 12;
      OPN   DI [LW 5];
      T     #LSQK.SCtrl;
      OPN   DI 2185;
      L     DIW 2;
      OPN   DI [LW 5];
      T     #LSQK.inRD;
      OPN   DI 2185;
      L     DIW 0;
      OPN   DI [LW 5];
      T     #LSQK.inRD_Statu;
      +AR2  P#4.0;
      UC    "HF3_LSQK_FB2522";
      LAR2  LD 1;
      L     #LSQK.qnWR;
      OPN   DI 2183;
      T     DIW 8;
      OPN   DI [LW 5];
      L     #LSQK.ToHMI;
      OPN   DI 6002;
      T     DIW 120;
      OPN   DI [LW 5];
      CDB;
      BLD   15;
      NOP   0;
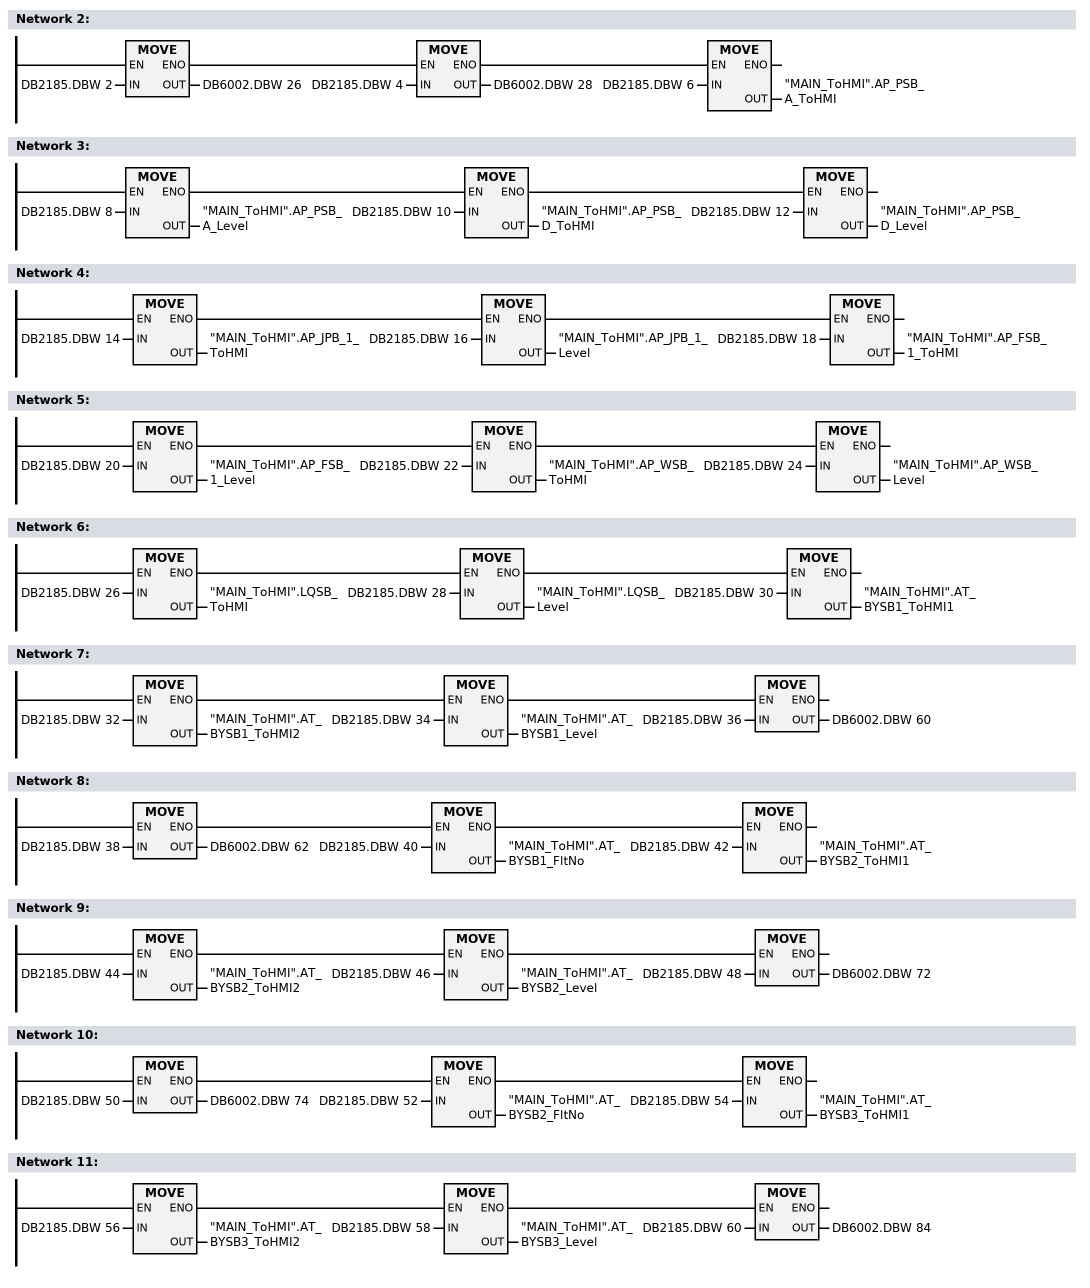
NETWORK
TITLE =
      A(;
      A(;
      L     DB2185.DBW 2;
      T     DB6002.DBW 26;
      SET;
      SAVE;
      CLR;
      A     BR;
      );
      JNB   _001;
      L     DB2185.DBW 4;
      T     DB6002.DBW 28;
      SET;
      SAVE;
      CLR;
_001: A     BR;
      );
      JNB   _002;
      L     DB2185.DBW 6;
      T     "MAIN_ToHMI".AP_PSB_A_ToHMI;
_002: NOP   0;
NETWORK
TITLE =
      A(;
      A(;
      L     DB2185.DBW 8;
      T     "MAIN_ToHMI".AP_PSB_A_Level;
      SET;
      SAVE;
      CLR;
      A     BR;
      );
      JNB   _003;
      L     DB2185.DBW 10;
      T     "MAIN_ToHMI".AP_PSB_D_ToHMI;
      SET;
      SAVE;
      CLR;
_003: A     BR;
      );
      JNB   _004;
      L     DB2185.DBW 12;
      T     "MAIN_ToHMI".AP_PSB_D_Level;
_004: NOP   0;
NETWORK
TITLE =
      A(;
      A(;
      L     DB2185.DBW 14;
      T     "MAIN_ToHMI".AP_JPB_1_ToHMI;
      SET;
      SAVE;
      CLR;
      A     BR;
      );
      JNB   _005;
      L     DB2185.DBW 16;
      T     "MAIN_ToHMI".AP_JPB_1_Level;
      SET;
      SAVE;
      CLR;
_005: A     BR;
      );
      JNB   _006;
      L     DB2185.DBW 18;
      T     "MAIN_ToHMI".AP_FSB_1_ToHMI;
_006: NOP   0;
NETWORK
TITLE =
      A(;
      A(;
      L     DB2185.DBW 20;
      T     "MAIN_ToHMI".AP_FSB_1_Level;
      SET;
      SAVE;
      CLR;
      A     BR;
      );
      JNB   _007;
      L     DB2185.DBW 22;
      T     "MAIN_ToHMI".AP_WSB_ToHMI;
      SET;
      SAVE;
      CLR;
_007: A     BR;
      );
      JNB   _008;
      L     DB2185.DBW 24;
      T     "MAIN_ToHMI".AP_WSB_Level;
_008: NOP   0;
NETWORK
TITLE =
      A(;
      A(;
      L     DB2185.DBW 26;
      T     "MAIN_ToHMI".LQSB_ToHMI;
      SET;
      SAVE;
      CLR;
      A     BR;
      );
      JNB   _009;
      L     DB2185.DBW 28;
      T     "MAIN_ToHMI".LQSB_Level;
      SET;
      SAVE;
      CLR;
_009: A     BR;
      );
      JNB   _00a;
      L     DB2185.DBW 30;
      T     "MAIN_ToHMI".AT_BYSB1_ToHMI1;
_00a: NOP   0;
NETWORK
TITLE =
      A(;
      A(;
      L     DB2185.DBW 32;
      T     "MAIN_ToHMI".AT_BYSB1_ToHMI2;
      SET;
      SAVE;
      CLR;
      A     BR;
      );
      JNB   _00b;
      L     DB2185.DBW 34;
      T     "MAIN_ToHMI".AT_BYSB1_Level;
      SET;
      SAVE;
      CLR;
_00b: A     BR;
      );
      JNB   _00c;
      L     DB2185.DBW 36;
      T     DB6002.DBW 60;
_00c: NOP   0;
NETWORK
TITLE =
      A(;
      A(;
      L     DB2185.DBW 38;
      T     DB6002.DBW 62;
      SET;
      SAVE;
      CLR;
      A     BR;
      );
      JNB   _00d;
      L     DB2185.DBW 40;
      T     "MAIN_ToHMI".AT_BYSB1_FltNo;
      SET;
      SAVE;
      CLR;
_00d: A     BR;
      );
      JNB   _00e;
      L     DB2185.DBW 42;
      T     "MAIN_ToHMI".AT_BYSB2_ToHMI1;
_00e: NOP   0;
NETWORK
TITLE =
      A(;
      A(;
      L     DB2185.DBW 44;
      T     "MAIN_ToHMI".AT_BYSB2_ToHMI2;
      SET;
      SAVE;
      CLR;
      A     BR;
      );
      JNB   _00f;
      L     DB2185.DBW 46;
      T     "MAIN_ToHMI".AT_BYSB2_Level;
      SET;
      SAVE;
      CLR;
_00f: A     BR;
      );
      JNB   _010;
      L     DB2185.DBW 48;
      T     DB6002.DBW 72;
_010: NOP   0;
NETWORK
TITLE =
      A(;
      A(;
      L     DB2185.DBW 50;
      T     DB6002.DBW 74;
      SET;
      SAVE;
      CLR;
      A     BR;
      );
      JNB   _011;
      L     DB2185.DBW 52;
      T     "MAIN_ToHMI".AT_BYSB2_FltNo;
      SET;
      SAVE;
      CLR;
_011: A     BR;
      );
      JNB   _012;
      L     DB2185.DBW 54;
      T     "MAIN_ToHMI".AT_BYSB3_ToHMI1;
_012: NOP   0;
NETWORK
TITLE =
      A(;
      A(;
      L     DB2185.DBW 56;
      T     "MAIN_ToHMI".AT_BYSB3_ToHMI2;
      SET;
      SAVE;
      CLR;
      A     BR;
      );
      JNB   _013;
      L     DB2185.DBW 58;
      T     "MAIN_ToHMI".AT_BYSB3_Level;
      SET;
      SAVE;
      CLR;
_013: A     BR;
      );
      JNB   _014;
      L     DB2185.DBW 60;
      T     DB6002.DBW 84;
_014: NOP   0;
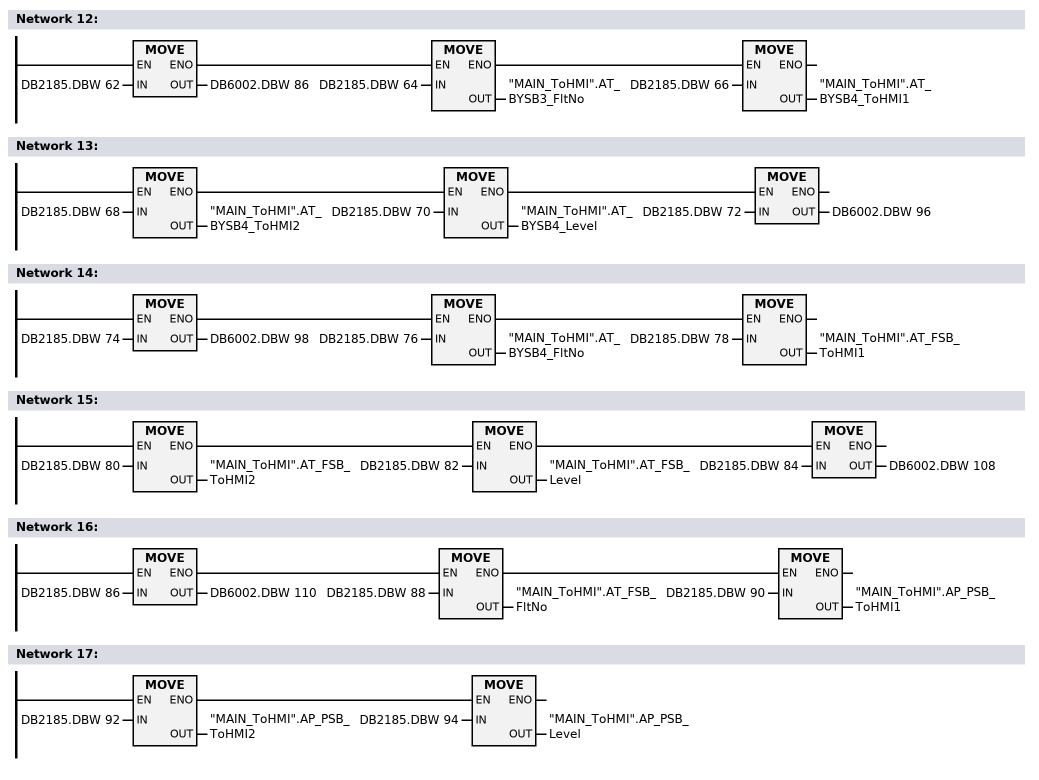
NETWORK
TITLE =
      A(;
      A(;
      L     DB2185.DBW 62;
      T     DB6002.DBW 86;
      SET;
      SAVE;
      CLR;
      A     BR;
      );
      JNB   _015;
      L     DB2185.DBW 64;
      T     "MAIN_ToHMI".AT_BYSB3_FltNo;
      SET;
      SAVE;
      CLR;
_015: A     BR;
      );
      JNB   _016;
      L     DB2185.DBW 66;
      T     "MAIN_ToHMI".AT_BYSB4_ToHMI1;
_016: NOP   0;
NETWORK
TITLE =
      A(;
      A(;
      L     DB2185.DBW 68;
      T     "MAIN_ToHMI".AT_BYSB4_ToHMI2;
      SET;
      SAVE;
      CLR;
      A     BR;
      );
      JNB   _017;
      L     DB2185.DBW 70;
      T     "MAIN_ToHMI".AT_BYSB4_Level;
      SET;
      SAVE;
      CLR;
_017: A     BR;
      );
      JNB   _018;
      L     DB2185.DBW 72;
      T     DB6002.DBW 96;
_018: NOP   0;
NETWORK
TITLE =
      A(;
      A(;
      L     DB2185.DBW 74;
      T     DB6002.DBW 98;
      SET;
      SAVE;
      CLR;
      A     BR;
      );
      JNB   _019;
      L     DB2185.DBW 76;
      T     "MAIN_ToHMI".AT_BYSB4_FltNo;
      SET;
      SAVE;
      CLR;
_019: A     BR;
      );
      JNB   _01a;
      L     DB2185.DBW 78;
      T     "MAIN_ToHMI".AT_FSB_ToHMI1;
_01a: NOP   0;
NETWORK
TITLE =
      A(;
      A(;
      L     DB2185.DBW 80;
      T     "MAIN_ToHMI".AT_FSB_ToHMI2;
      SET;
      SAVE;
      CLR;
      A     BR;
      );
      JNB   _01b;
      L     DB2185.DBW 82;
      T     "MAIN_ToHMI".AT_FSB_Level;
      SET;
      SAVE;
      CLR;
_01b: A     BR;
      );
      JNB   _01c;
      L     DB2185.DBW 84;
      T     DB6002.DBW 108;
_01c: NOP   0;
NETWORK
TITLE =
      A(;
      A(;
      L     DB2185.DBW 86;
      T     DB6002.DBW 110;
      SET;
      SAVE;
      CLR;
      A     BR;
      );
      JNB   _01d;
      L     DB2185.DBW 88;
      T     "MAIN_ToHMI".AT_FSB_FltNo;
      SET;
      SAVE;
      CLR;
_01d: A     BR;
      );
      JNB   _01e;
      L     DB2185.DBW 90;
      T     "MAIN_ToHMI".AP_PSB_ToHMI1;
_01e: NOP   0;
NETWORK
TITLE =
      A(;
      L     DB2185.DBW 92;
      T     "MAIN_ToHMI".AP_PSB_ToHMI2;
      SET;
      SAVE;
      CLR;
      A     BR;
      );
      JNB   _01f;
      L     DB2185.DBW 94;
      T     "MAIN_ToHMI".AP_PSB_Level;
_01f: NOP   0;
END_FUNCTION_BLOCK

FUNCTION_BLOCK "HF3_LSQK_FB2522"	// FB 2522
VERSION : 0.1
VAR_INPUT
  SCtrl : WORD ;
  inRD : WORD ;	//读取值
  inRD_Statu : WORD ;	//通信状态
  Heat_Load_Set : INT ;	//公共区热符合设定
  Station_C_Set : INT ;	//站厅温度设定
  Platform_C_Set : INT ;	//站台温度设定
  H_P_All_Ctrl : WORD ;	//全局控制命令
  FireAlarm : BOOL ;	//火灾信息
  PT : TIME ;	//超时时间
END_VAR
VAR_OUTPUT
  qnWR : WORD ;	//输出控制信息
  ToHMI : WORD ;
END_VAR
VAR
  Ton1 : SFB 4;
  Ton2 : SFB 4;
  SCtrl_Temp : ARRAY  [0 .. 15 ] OF //0-启动控制1-停止控制
  BOOL ;
  Ctrl : ARRAY  [0 .. 1 ] OF //0-启动控制1-停止控制
  BOOL ;
  Latch : ARRAY  [0 .. 1 ] OF //0-启动控制锁定1-停止控制锁定
  BOOL ;
  DI_Temp : ARRAY  [0 .. 15 ] OF //8-远程状态9-总故障信息
  BOOL ;
  DO_Temp : ARRAY  [0 .. 15 ] OF //8-启动9-停止
  BOOL ;
  SIngTout : BOOL ;	//输入超时
  QTout : BOOL ;	//输出超时
  Timeout : BOOL ;	//超时时间
  McFlag : BOOL ;	//检修牌
  H_P_All_Ctrl_Temp : ARRAY  [0 .. 15 ] OF //全局命令
  BOOL ;
  CommOK : BOOL ;
END_VAR
BEGIN
NETWORK
TITLE =
      A(;
      BLD   1;
      =     L 4.0;
      TAR2  LD 0;
      L     #SCtrl;
      T     LW 5;
      L     DINO;
      T     LW 7;
      +AR2  P#68.0;
      TAR2;
      LAR2  LD 0;
      T     LD 9;
      UC    "HF3_W_T_B_FC54";
      {     P#L 5.0, P#L 7.0 };
      LAR2  LD 0;
      BLD   2;
      A     BR;
      );
      JNB   _001;
      BLD   1;
      =     L 4.0;
      TAR2  LD 0;
      L     #H_P_All_Ctrl;
      T     LW 5;
      L     DINO;
      T     LW 7;
      +AR2  P#80.0;
      TAR2;
      LAR2  LD 0;
      T     LD 9;
      UC    "HF3_W_T_B_FC54";
      {     P#L 5.0, P#L 7.0 };
      LAR2  LD 0;
      BLD   2;
_001: NOP   0;
NETWORK
TITLE =
      BLD   1;
      =     L 4.0;
      TAR2  LD 0;
      L     #inRD;
      T     LW 5;
      L     DINO;
      T     LW 7;
      +AR2  P#74.0;
      TAR2;
      LAR2  LD 0;
      T     LD 9;
      UC    "HF3_W_T_B_FC54";
      {     P#L 5.0, P#L 7.0 };
      LAR2  LD 0;
      BLD   2;
      NOP   0;
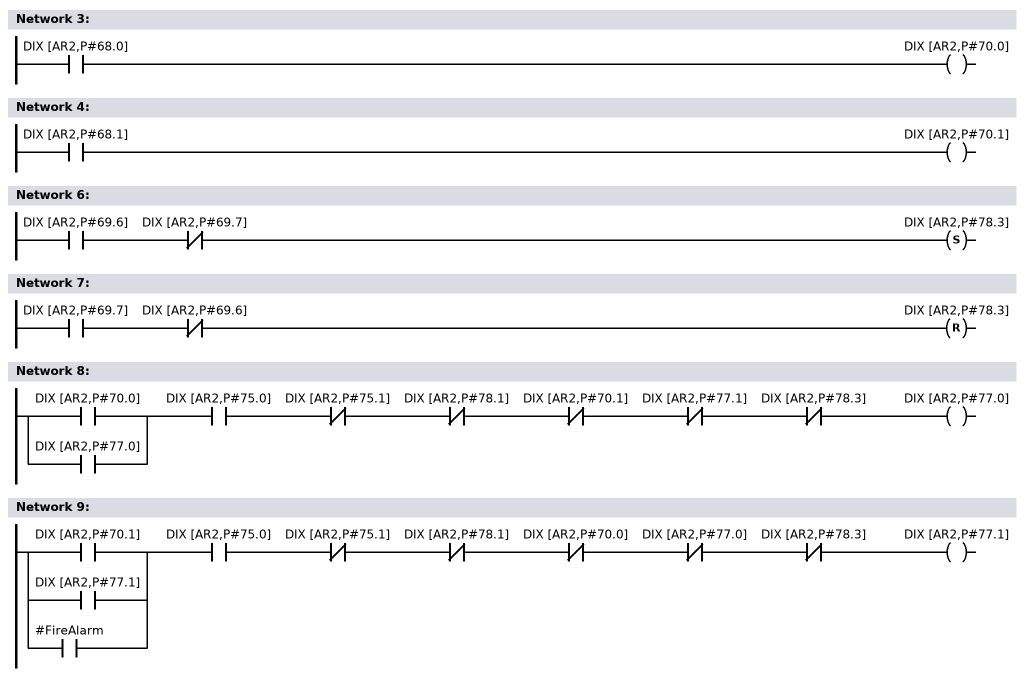
NETWORK
TITLE =
      A     DIX [AR2,P#68.0];
      =     DIX [AR2,P#70.0];
NETWORK
TITLE =
      A     DIX [AR2,P#68.1];
      =     DIX [AR2,P#70.1];
NETWORK
TITLE =
      A(;
      O     DIX [AR2,P#77.0];
      O     DIX [AR2,P#77.1];
      );
      =     L 0.0;
      BLD   103;
      BLD   16;
      =     L 7.0;
      L     DINO;
      T     LW 5;
      CDB;
      OPN   DI [LW 5];
      TAR2  LD 1;
      A     L 0.0;
      =     DIX [AR2,P#24.0];
      L     DBD [AR2,P#16.0];
      T     DID [AR2,P#26.0];
      +AR2  P#24.0;
      UC    "TON";
      LAR2  LD 1;
      A     DIX [AR2,P#30.0];
      =     DBX [AR2,P#78.1];
      CDB;
      BLD   17;
      NOP   0;
NETWORK
TITLE =
      A     DIX [AR2,P#69.6];
      AN    DIX [AR2,P#69.7];
      S     DIX [AR2,P#78.3];
NETWORK
TITLE =
      A     DIX [AR2,P#69.7];
      AN    DIX [AR2,P#69.6];
      R     DIX [AR2,P#78.3];
NETWORK
TITLE =
      A(;
      O     DIX [AR2,P#70.0];
      O     DIX [AR2,P#77.0];
      );
      A     DIX [AR2,P#75.0];
      AN    DIX [AR2,P#75.1];
      AN    DIX [AR2,P#78.1];
      AN    DIX [AR2,P#70.1];
      AN    DIX [AR2,P#77.1];
      AN    DIX [AR2,P#78.3];
      =     DIX [AR2,P#77.0];
NETWORK
TITLE =
      A(;
      O     DIX [AR2,P#70.1];
      O     DIX [AR2,P#77.1];
      O     #FireAlarm;
      );
      A     DIX [AR2,P#75.0];
      AN    DIX [AR2,P#75.1];
      AN    DIX [AR2,P#78.1];
      AN    DIX [AR2,P#70.0];
      AN    DIX [AR2,P#77.0];
      AN    DIX [AR2,P#78.3];
      =     DIX [AR2,P#77.1];
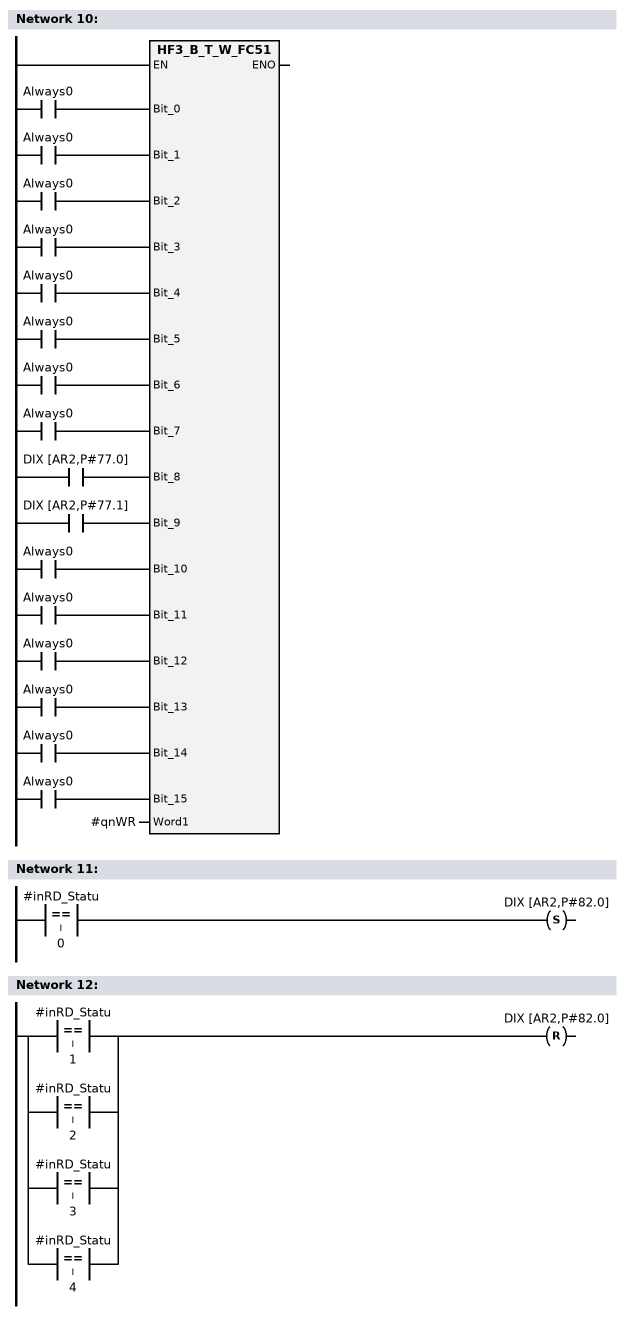
NETWORK
TITLE =
      A     "Always0";
      =     L 0.0;
      BLD   103;
      A     "Always0";
      =     L 0.1;
      BLD   103;
      A     "Always0";
      =     L 0.2;
      BLD   103;
      A     "Always0";
      =     L 0.3;
      BLD   103;
      A     "Always0";
      =     L 0.4;
      BLD   103;
      A     "Always0";
      =     L 0.5;
      BLD   103;
      A     "Always0";
      =     L 0.6;
      BLD   103;
      A     "Always0";
      =     L 0.7;
      BLD   103;
      A     DIX [AR2,P#77.0];
      =     L 1.0;
      BLD   103;
      A     DIX [AR2,P#77.1];
      =     L 1.1;
      BLD   103;
      A     "Always0";
      =     L 1.2;
      BLD   103;
      A     "Always0";
      =     L 1.3;
      BLD   103;
      A     "Always0";
      =     L 1.4;
      BLD   103;
      A     "Always0";
      =     L 1.5;
      BLD   103;
      A     "Always0";
      =     L 1.6;
      BLD   103;
      A     "Always0";
      =     L 1.7;
      BLD   103;
      CALL  "HF3_B_T_W_FC51" (
           Bit_0                    := L 0.0,
           Bit_1                    := L 0.1,
           Bit_2                    := L 0.2,
           Bit_3                    := L 0.3,
           Bit_4                    := L 0.4,
           Bit_5                    := L 0.5,
           Bit_6                    := L 0.6,
           Bit_7                    := L 0.7,
           Bit_8                    := L 1.0,
           Bit_9                    := L 1.1,
           Bit_10                   := L 1.2,
           Bit_11                   := L 1.3,
           Bit_12                   := L 1.4,
           Bit_13                   := L 1.5,
           Bit_14                   := L 1.6,
           Bit_15                   := L 1.7,
           Word1                    := #qnWR);
      NOP   0;
NETWORK
TITLE =
      L     #inRD_Statu;
      L     0;
      ==I;
      S     DIX [AR2,P#82.0];
NETWORK
TITLE =
      O(;
      L     #inRD_Statu;
      L     1;
      ==I;
      );
      O(;
      L     #inRD_Statu;
      L     2;
      ==I;
      );
      O(;
      L     #inRD_Statu;
      L     3;
      ==I;
      );
      O(;
      L     #inRD_Statu;
      L     4;
      ==I;
      );
      R     DIX [AR2,P#82.0];
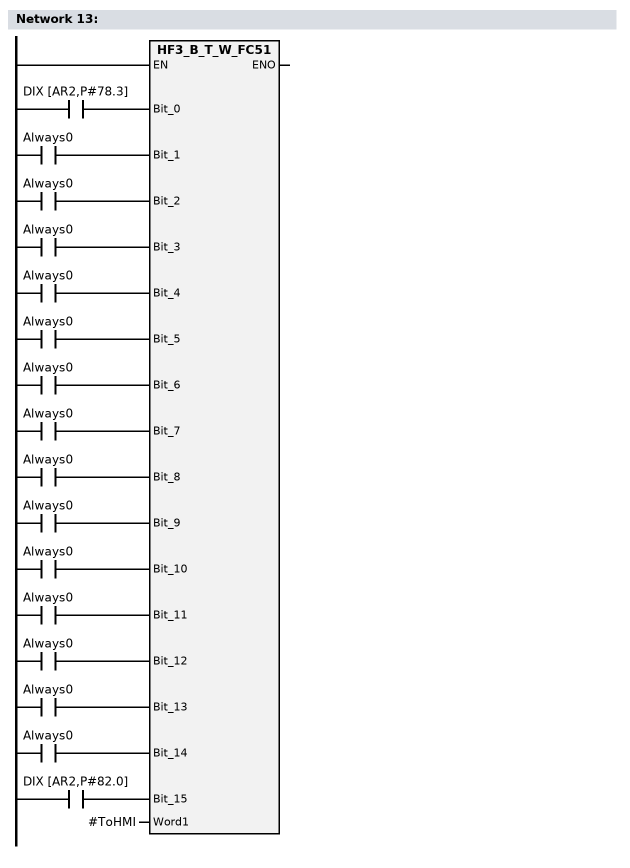
NETWORK
TITLE =
      A     DIX [AR2,P#78.3];
      =     L 0.0;
      BLD   103;
      A     "Always0";
      =     L 0.1;
      BLD   103;
      A     "Always0";
      =     L 0.2;
      BLD   103;
      A     "Always0";
      =     L 0.3;
      BLD   103;
      A     "Always0";
      =     L 0.4;
      BLD   103;
      A     "Always0";
      =     L 0.5;
      BLD   103;
      A     "Always0";
      =     L 0.6;
      BLD   103;
      A     "Always0";
      =     L 0.7;
      BLD   103;
      A     "Always0";
      =     L 1.0;
      BLD   103;
      A     "Always0";
      =     L 1.1;
      BLD   103;
      A     "Always0";
      =     L 1.2;
      BLD   103;
      A     "Always0";
      =     L 1.3;
      BLD   103;
      A     "Always0";
      =     L 1.4;
      BLD   103;
      A     "Always0";
      =     L 1.5;
      BLD   103;
      A     "Always0";
      =     L 1.6;
      BLD   103;
      A     DIX [AR2,P#82.0];
      =     L 1.7;
      BLD   103;
      CALL  "HF3_B_T_W_FC51" (
           Bit_0                    := L 0.0,
           Bit_1                    := L 0.1,
           Bit_2                    := L 0.2,
           Bit_3                    := L 0.3,
           Bit_4                    := L 0.4,
           Bit_5                    := L 0.5,
           Bit_6                    := L 0.6,
           Bit_7                    := L 0.7,
           Bit_8                    := L 1.0,
           Bit_9                    := L 1.1,
           Bit_10                   := L 1.2,
           Bit_11                   := L 1.3,
           Bit_12                   := L 1.4,
           Bit_13                   := L 1.5,
           Bit_14                   := L 1.6,
           Bit_15                   := L 1.7,
           Word1                    := #ToHMI);
      NOP   0;
END_FUNCTION_BLOCK

FUNCTION_BLOCK "HF3_JET_FB2531"	// FB 2531
TITLE = 处理车站该端射流风机
VERSION : 0.1
VAR
  JET_1 : FB 2532;
  JET_2 : FB 2532;
END_VAR
BEGIN
NETWORK
TITLE = 同一台控制柜包含两台风机
      A(;
      A     M 42.0;
      =     L 0.3;
      BLD   103;
      A     M 42.1;
      =     L 0.4;
      BLD   103;
      A     M 42.2;
      =     L 0.5;
      BLD   103;
      BLD   14;
      =     L 7.0;
      L     DINO;
      T     LW 5;
      CDB;
      OPN   DI [LW 5];
      TAR2  LD 1;
      L     MW 34;
      T     #JET_1.SCtrl1;
      L     MW 38;
      T     #JET_1.inRD;
      L     L#20000;
      T     #JET_1.PT2;
      A     L 0.3;
      =     #JET_1.Open;
      A     L 0.4;
      =     #JET_1.FireAlarm;
      A     L 0.5;
      =     #JET_1.BlockAlarm;
      +AR2  P#0.0;
      UC    "HF3_JET_FB2532";
      LAR2  LD 1;
      L     #JET_1.qnWR;
      T     MW 60;
      CDB;
      BLD   15;
      A     BR;
      );
      JNB   _001;
      BLD   14;
      =     L 7.0;
      L     DINO;
      T     LW 5;
      CDB;
      OPN   DI [LW 5];
      TAR2  LD 1;
      L     L#20000;
      T     DID [AR2,P#124.0];
      +AR2  P#118.0;
      UC    "HF3_JET_FB2532";
      LAR2  LD 1;
      CDB;
      BLD   15;
_001: NOP   0;
NETWORK
TITLE =
END_FUNCTION_BLOCK

FUNCTION_BLOCK "HF3_JET_FB2532"	// FB 2532
VERSION : 0.1
VAR_INPUT
  SCtrl1 : WORD ;	//上位控制命令
  SCtrl2 : WORD ;
  inRD : WORD ;	//输入状态字
  PT2 : TIME ;	//超时时间
  H_P_ALL_Ctrl : WORD ;	//全局控制命令
  MCtrl : ARRAY  [0 .. 3 ] OF //0-正转1-反转2-停止
  BOOL ;
  Mode : ARRAY  [0 .. 15 ] OF //0-开始1-结束2-执行中
  BOOL ;
  Open : BOOL ;	//风机联锁开
  ALL : ARRAY  [0 .. 15 ] OF //0-单控1-模控2-时间表
  BOOL ;
  FireAlarm : BOOL ;	//火灾模式
  BlockAlarm : BOOL ;	//阻塞模式
END_VAR
VAR_OUTPUT
  qnWR : WORD ;	//控制命令
  ToHMI : WORD ;	//反馈上位信息1
  RT : INT ;	//1风机运行时间
  SumFlt : INT ;	//1风机故障次数
  SumRun : INT ;	//1风机运行次数
  Refuse : BOOL ;
END_VAR
VAR
  Ton1 : SFB 4;
  Ton2 : SFB 4;
  Ton3 : SFB 4;
  SFlag : BOOL ;	//单控标志
  SingTout : BOOL ;	//控制命令超时
  Timeout : BOOL ;	//风机超时
  DI_Temp : ARRAY  [0 .. 15 ] OF //01-按钮23-正反运行4-停止
  BOOL ;
  DO_Temp : ARRAY  [0 .. 15 ] OF //01-1正反转23-2火灾正反转4-停止
  BOOL ;
  Ctrl : ARRAY  [0 .. 15 ] OF //01-1正反转23-2火灾正反转4-停止
  BOOL ;
  SCtrl_Temp1 : ARRAY  [0 .. 15 ] OF //01-单模控 23-正反转 45-正反转 6-停
  BOOL ;
  Latch : ARRAY  [0 .. 7 ] OF //01-正反转锁定23-2火灾正反转
  BOOL ;
  McFlag : BOOL ;	//挂检修牌
  QTout : BOOL ;	//输出超时
  H_P_ALL_Ctrl_Temp : ARRAY  [0 .. 15 ] OF BOOL ;
  Ctrl_En1 : BOOL ;	//正常启动使能
  Ctrl_En2 : BOOL ;	//火灾启动使能
  CommOK : BOOL ;	//通信正常
END_VAR
BEGIN
NETWORK
TITLE =
      A(;
      BLD   1;
      =     L 4.0;
      TAR2  LD 0;
      L     #SCtrl1;
      T     LW 5;
      L     DINO;
      T     LW 7;
      +AR2  P#108.0;
      TAR2;
      LAR2  LD 0;
      T     LD 9;
      UC    "HF3_W_T_B_FC54";
      {     P#L 5.0, P#L 7.0 };
      LAR2  LD 0;
      BLD   2;
      A     BR;
      );
      JNB   _001;
      BLD   1;
      =     L 4.0;
      TAR2  LD 0;
      L     #H_P_ALL_Ctrl;
      T     LW 5;
      L     DINO;
      T     LW 7;
      +AR2  P#114.0;
      TAR2;
      LAR2  LD 0;
      T     LD 9;
      UC    "HF3_W_T_B_FC54";
      {     P#L 5.0, P#L 7.0 };
      LAR2  LD 0;
      BLD   2;
_001: NOP   0;
NETWORK
TITLE =  
      BLD   1;
      =     L 4.0;
      TAR2  LD 0;
      L     #inRD;
      T     LW 5;
      L     DINO;
      T     LW 7;
      +AR2  P#102.0;
      TAR2;
      LAR2  LD 0;
      T     LD 9;
      UC    "HF3_W_T_B_FC54";
      {     P#L 5.0, P#L 7.0 };
      LAR2  LD 0;
      BLD   2;
      NOP   0;
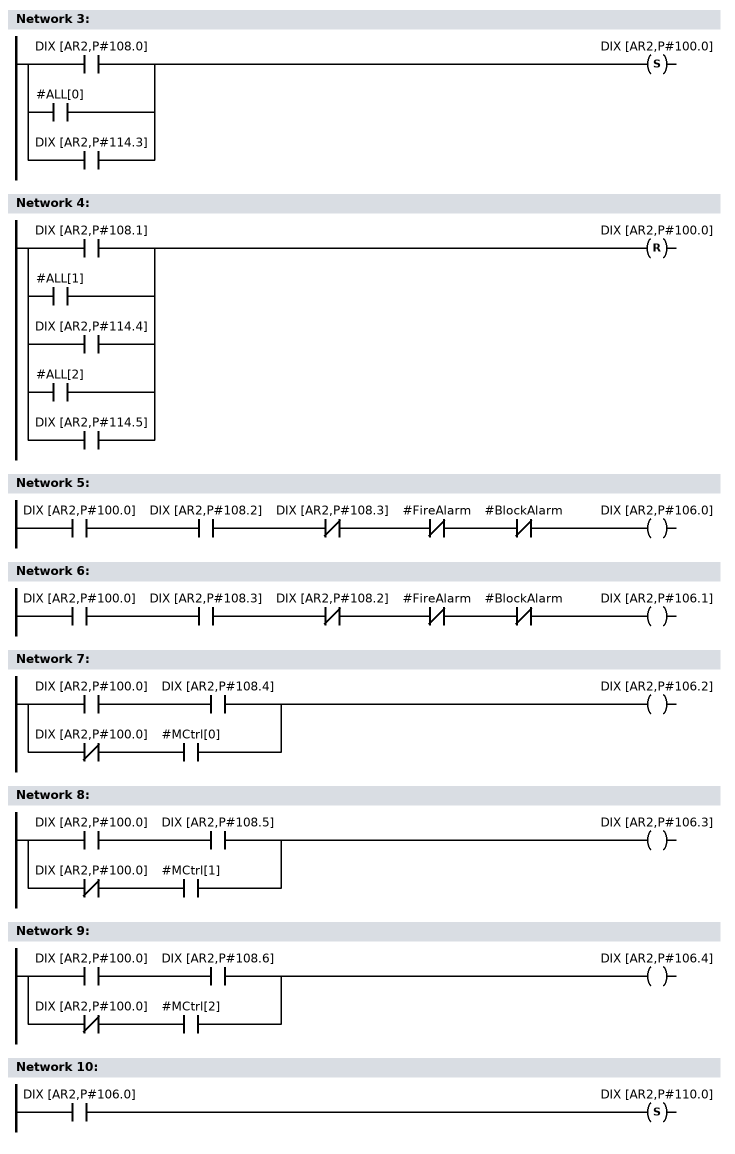
NETWORK
TITLE =
      O     DIX [AR2,P#108.0];
      O     #ALL[0];
      O     DIX [AR2,P#114.3];
      S     DIX [AR2,P#100.0];
NETWORK
TITLE =
      O     DIX [AR2,P#108.1];
      O     #ALL[1];
      O     DIX [AR2,P#114.4];
      O     #ALL[2];
      O     DIX [AR2,P#114.5];
      R     DIX [AR2,P#100.0];
NETWORK
TITLE =
      A     DIX [AR2,P#100.0];
      A     DIX [AR2,P#108.2];
      AN    DIX [AR2,P#108.3];
      AN    #FireAlarm;
      AN    #BlockAlarm;
      =     DIX [AR2,P#106.0];
NETWORK
TITLE =
      A     DIX [AR2,P#100.0];
      A     DIX [AR2,P#108.3];
      AN    DIX [AR2,P#108.2];
      AN    #FireAlarm;
      AN    #BlockAlarm;
      =     DIX [AR2,P#106.1];
NETWORK
TITLE =
      A     DIX [AR2,P#100.0];
      A     DIX [AR2,P#108.4];
      O;
      AN    DIX [AR2,P#100.0];
      A     #MCtrl[0];
      =     DIX [AR2,P#106.2];
NETWORK
TITLE =
      A     DIX [AR2,P#100.0];
      A     DIX [AR2,P#108.5];
      O;
      AN    DIX [AR2,P#100.0];
      A     #MCtrl[1];
      =     DIX [AR2,P#106.3];
NETWORK
TITLE =
      A     DIX [AR2,P#100.0];
      A     DIX [AR2,P#108.6];
      O;
      AN    DIX [AR2,P#100.0];
      A     #MCtrl[2];
      =     DIX [AR2,P#106.4];
NETWORK
TITLE =
      A     DIX [AR2,P#106.0];
      S     DIX [AR2,P#110.0];
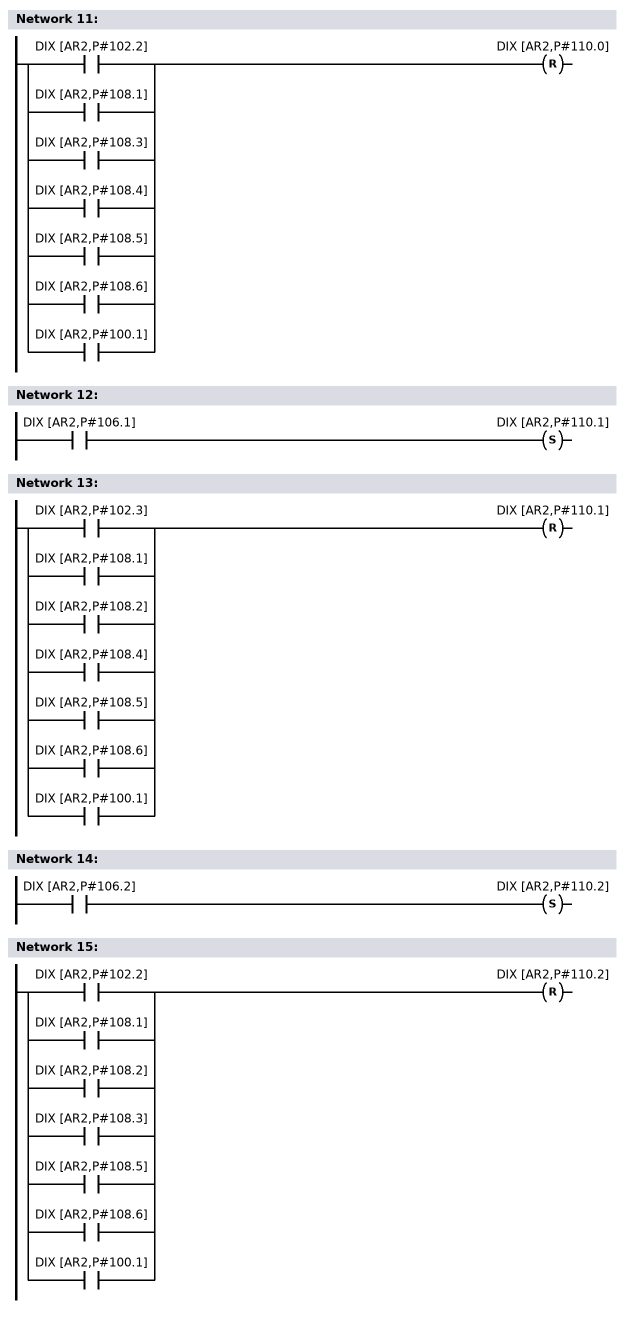
NETWORK
TITLE =
      O     DIX [AR2,P#102.2];
      O     DIX [AR2,P#108.1];
      O     DIX [AR2,P#108.3];
      O     DIX [AR2,P#108.4];
      O     DIX [AR2,P#108.5];
      O     DIX [AR2,P#108.6];
      O     DIX [AR2,P#100.1];
      R     DIX [AR2,P#110.0];
NETWORK
TITLE =
      A     DIX [AR2,P#106.1];
      S     DIX [AR2,P#110.1];
NETWORK
TITLE =
      O     DIX [AR2,P#102.3];
      O     DIX [AR2,P#108.1];
      O     DIX [AR2,P#108.2];
      O     DIX [AR2,P#108.4];
      O     DIX [AR2,P#108.5];
      O     DIX [AR2,P#108.6];
      O     DIX [AR2,P#100.1];
      R     DIX [AR2,P#110.1];
NETWORK
TITLE =
      A     DIX [AR2,P#106.2];
      S     DIX [AR2,P#110.2];
NETWORK
TITLE =
      O     DIX [AR2,P#102.2];
      O     DIX [AR2,P#108.1];
      O     DIX [AR2,P#108.2];
      O     DIX [AR2,P#108.3];
      O     DIX [AR2,P#108.5];
      O     DIX [AR2,P#108.6];
      O     DIX [AR2,P#100.1];
      R     DIX [AR2,P#110.2];
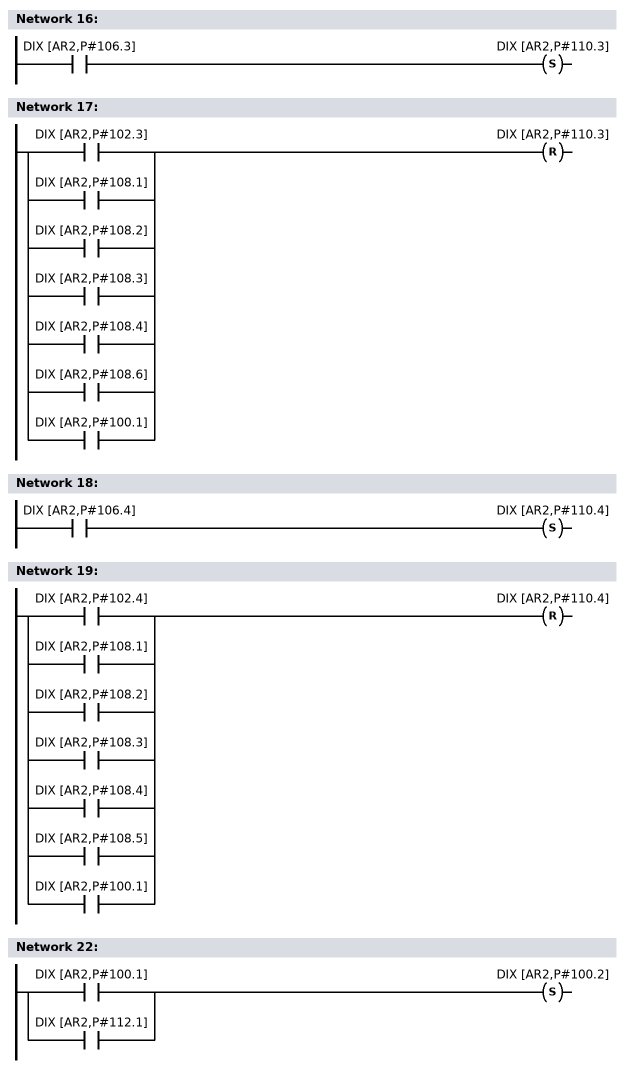
NETWORK
TITLE =
      A     DIX [AR2,P#106.3];
      S     DIX [AR2,P#110.3];
NETWORK
TITLE =
      O     DIX [AR2,P#102.3];
      O     DIX [AR2,P#108.1];
      O     DIX [AR2,P#108.2];
      O     DIX [AR2,P#108.3];
      O     DIX [AR2,P#108.4];
      O     DIX [AR2,P#108.6];
      O     DIX [AR2,P#100.1];
      R     DIX [AR2,P#110.3];
NETWORK
TITLE =
      A     DIX [AR2,P#106.4];
      S     DIX [AR2,P#110.4];
NETWORK
TITLE =
      O     DIX [AR2,P#102.4];
      O     DIX [AR2,P#108.1];
      O     DIX [AR2,P#108.2];
      O     DIX [AR2,P#108.3];
      O     DIX [AR2,P#108.4];
      O     DIX [AR2,P#108.5];
      O     DIX [AR2,P#100.1];
      R     DIX [AR2,P#110.4];
NETWORK
TITLE =
      A(;
      O     DIX [AR2,P#110.0];
      O     DIX [AR2,P#110.1];
      O     DIX [AR2,P#110.2];
      O     DIX [AR2,P#110.3];
      );
      =     L 0.0;
      BLD   103;
      BLD   16;
      =     L 7.0;
      L     DINO;
      T     LW 5;
      CDB;
      OPN   DI [LW 5];
      TAR2  LD 1;
      A     L 0.0;
      =     DIX [AR2,P#34.0];
      L     DBD [AR2,P#6.0];
      T     DID [AR2,P#36.0];
      +AR2  P#34.0;
      UC    "TON";
      LAR2  LD 1;
      A     DIX [AR2,P#40.0];
      =     DBX [AR2,P#100.1];
      CDB;
      BLD   17;
      NOP   0;
NETWORK
TITLE =
      A(;
      O     DIX [AR2,P#104.0];
      O     DIX [AR2,P#104.1];
      O     DIX [AR2,P#104.2];
      O     DIX [AR2,P#104.3];
      O     DIX [AR2,P#104.4];
      );
      =     L 0.0;
      BLD   103;
      BLD   16;
      =     L 7.0;
      L     DINO;
      T     LW 5;
      CDB;
      OPN   DI [LW 5];
      TAR2  LD 1;
      A     L 0.0;
      =     DIX [AR2,P#56.0];
      L     DBD [AR2,P#6.0];
      T     DID [AR2,P#58.0];
      +AR2  P#56.0;
      UC    "TON";
      LAR2  LD 1;
      A     DIX [AR2,P#62.0];
      =     DBX [AR2,P#112.1];
      CDB;
      BLD   17;
      NOP   0;
NETWORK
TITLE =
      O     DIX [AR2,P#100.1];
      O     DIX [AR2,P#112.1];
      S     DIX [AR2,P#100.2];
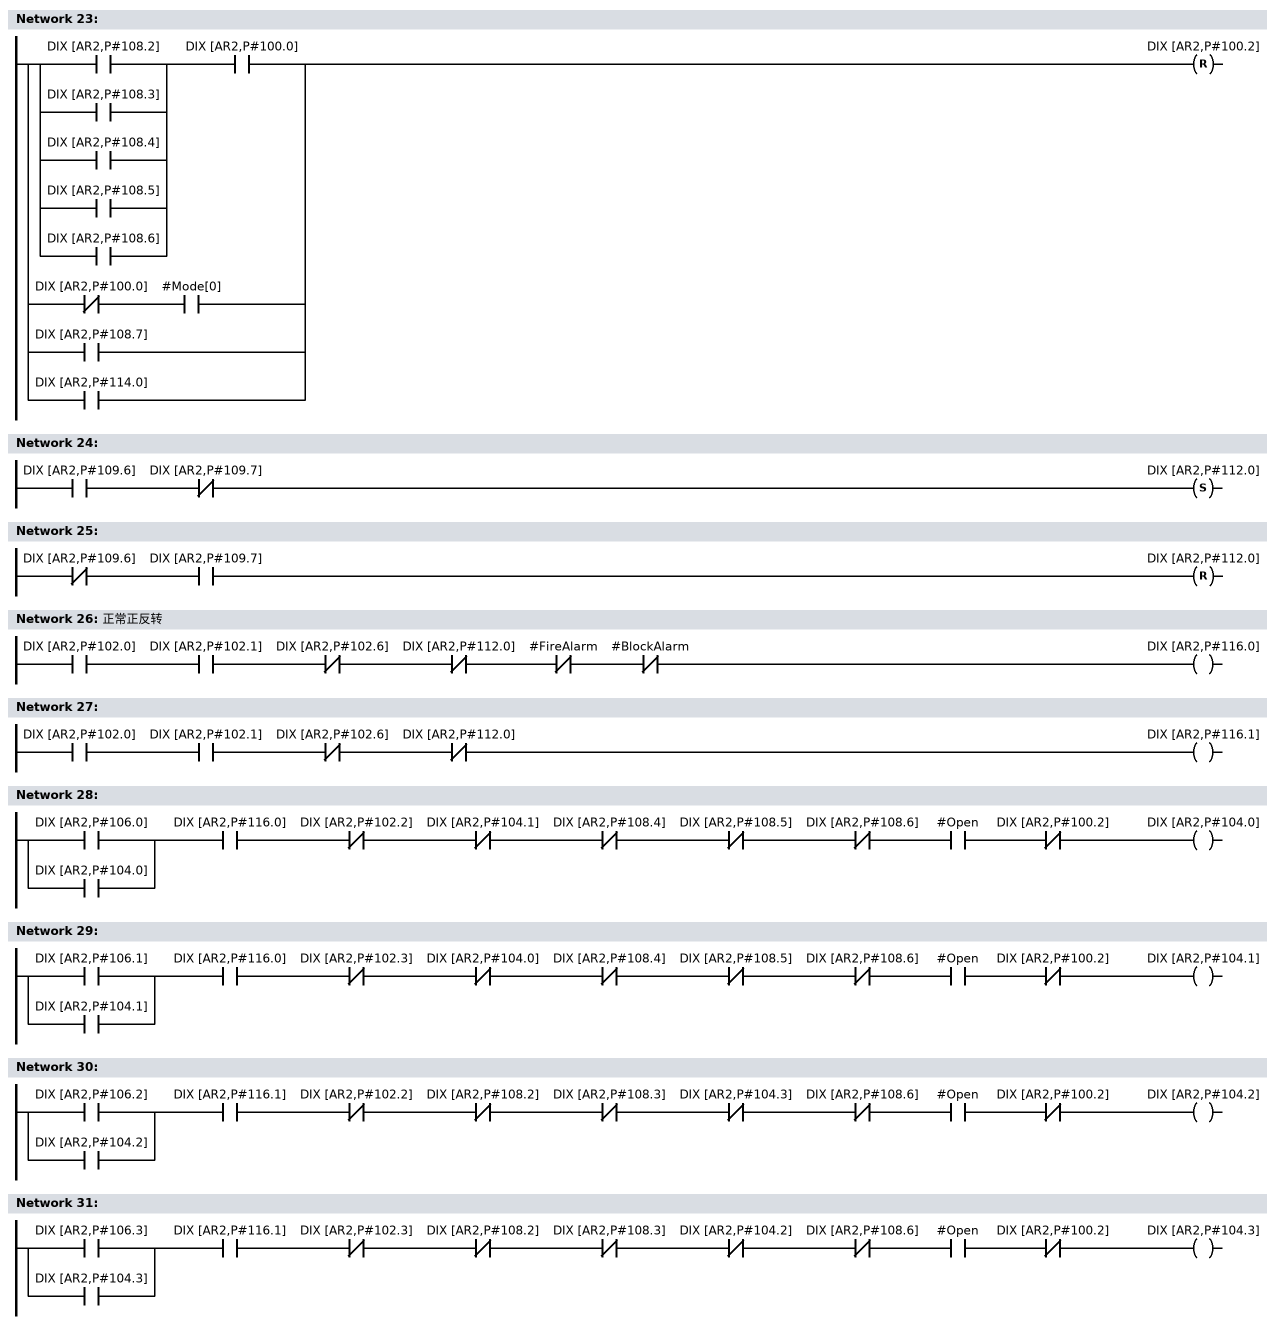
NETWORK
TITLE =
      A(;
      O     DIX [AR2,P#108.2];
      O     DIX [AR2,P#108.3];
      O     DIX [AR2,P#108.4];
      O     DIX [AR2,P#108.5];
      O     DIX [AR2,P#108.6];
      );
      A     DIX [AR2,P#100.0];
      O;
      AN    DIX [AR2,P#100.0];
      A     #Mode[0];
      O     DIX [AR2,P#108.7];
      O     DIX [AR2,P#114.0];
      R     DIX [AR2,P#100.2];
NETWORK
TITLE =
      A     DIX [AR2,P#109.6];
      AN    DIX [AR2,P#109.7];
      S     DIX [AR2,P#112.0];
NETWORK
TITLE =
      AN    DIX [AR2,P#109.6];
      A     DIX [AR2,P#109.7];
      R     DIX [AR2,P#112.0];
NETWORK
TITLE = 正常正反转
      A     DIX [AR2,P#102.0];
      A     DIX [AR2,P#102.1];
      AN    DIX [AR2,P#102.6];
      AN    DIX [AR2,P#112.0];
      AN    #FireAlarm;
      AN    #BlockAlarm;
      =     DIX [AR2,P#116.0];
NETWORK
TITLE =
      A     DIX [AR2,P#102.0];
      A     DIX [AR2,P#102.1];
      AN    DIX [AR2,P#102.6];
      AN    DIX [AR2,P#112.0];
      =     DIX [AR2,P#116.1];
NETWORK
TITLE =
      A(;
      O     DIX [AR2,P#106.0];
      O     DIX [AR2,P#104.0];
      );
      A     DIX [AR2,P#116.0];
      AN    DIX [AR2,P#102.2];
      AN    DIX [AR2,P#104.1];
      AN    DIX [AR2,P#108.4];
      AN    DIX [AR2,P#108.5];
      AN    DIX [AR2,P#108.6];
      A     #Open;
      AN    DIX [AR2,P#100.2];
      =     DIX [AR2,P#104.0];
NETWORK
TITLE =
      A(;
      O     DIX [AR2,P#106.1];
      O     DIX [AR2,P#104.1];
      );
      A     DIX [AR2,P#116.0];
      AN    DIX [AR2,P#102.3];
      AN    DIX [AR2,P#104.0];
      AN    DIX [AR2,P#108.4];
      AN    DIX [AR2,P#108.5];
      AN    DIX [AR2,P#108.6];
      A     #Open;
      AN    DIX [AR2,P#100.2];
      =     DIX [AR2,P#104.1];
NETWORK
TITLE =
      A(;
      O     DIX [AR2,P#106.2];
      O     DIX [AR2,P#104.2];
      );
      A     DIX [AR2,P#116.1];
      AN    DIX [AR2,P#102.2];
      AN    DIX [AR2,P#108.2];
      AN    DIX [AR2,P#108.3];
      AN    DIX [AR2,P#104.3];
      AN    DIX [AR2,P#108.6];
      A     #Open;
      AN    DIX [AR2,P#100.2];
      =     DIX [AR2,P#104.2];
NETWORK
TITLE =
      A(;
      O     DIX [AR2,P#106.3];
      O     DIX [AR2,P#104.3];
      );
      A     DIX [AR2,P#116.1];
      AN    DIX [AR2,P#102.3];
      AN    DIX [AR2,P#108.2];
      AN    DIX [AR2,P#108.3];
      AN    DIX [AR2,P#104.2];
      AN    DIX [AR2,P#108.6];
      A     #Open;
      AN    DIX [AR2,P#100.2];
      =     DIX [AR2,P#104.3];
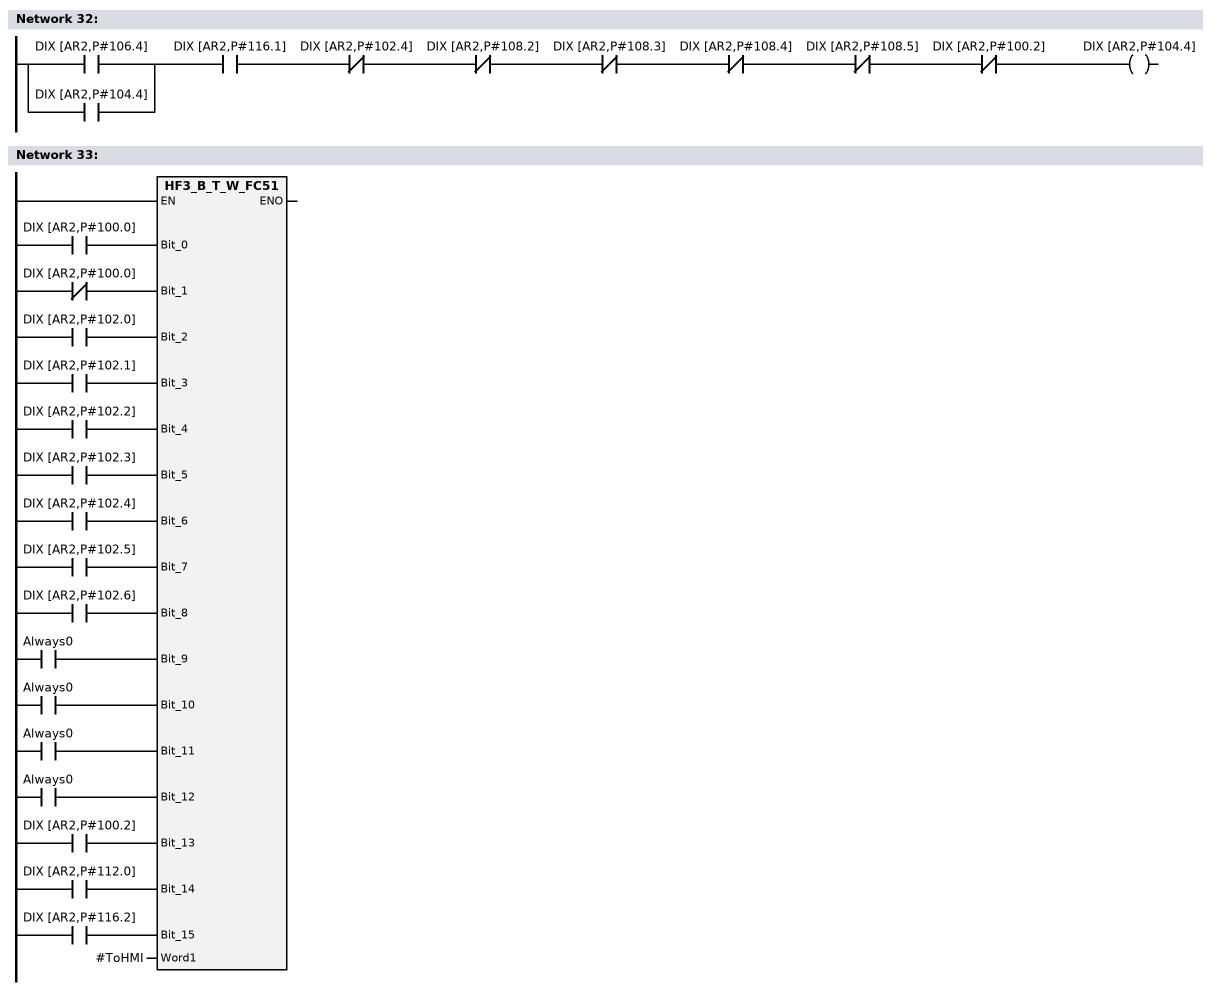
NETWORK
TITLE =
      A(;
      O     DIX [AR2,P#106.4];
      O     DIX [AR2,P#104.4];
      );
      A     DIX [AR2,P#116.1];
      AN    DIX [AR2,P#102.4];
      AN    DIX [AR2,P#108.2];
      AN    DIX [AR2,P#108.3];
      AN    DIX [AR2,P#108.4];
      AN    DIX [AR2,P#108.5];
      AN    DIX [AR2,P#100.2];
      =     DIX [AR2,P#104.4];
NETWORK
TITLE =
      A     DIX [AR2,P#100.0];
      =     L 0.0;
      BLD   103;
      AN    DIX [AR2,P#100.0];
      =     L 0.1;
      BLD   103;
      A     DIX [AR2,P#102.0];
      =     L 0.2;
      BLD   103;
      A     DIX [AR2,P#102.1];
      =     L 0.3;
      BLD   103;
      A     DIX [AR2,P#102.2];
      =     L 0.4;
      BLD   103;
      A     DIX [AR2,P#102.3];
      =     L 0.5;
      BLD   103;
      A     DIX [AR2,P#102.4];
      =     L 0.6;
      BLD   103;
      A     DIX [AR2,P#102.5];
      =     L 0.7;
      BLD   103;
      A     DIX [AR2,P#102.6];
      =     L 1.0;
      BLD   103;
      A     "Always0";
      =     L 1.1;
      BLD   103;
      A     "Always0";
      =     L 1.2;
      BLD   103;
      A     "Always0";
      =     L 1.3;
      BLD   103;
      A     "Always0";
      =     L 1.4;
      BLD   103;
      A     DIX [AR2,P#100.2];
      =     L 1.5;
      BLD   103;
      A     DIX [AR2,P#112.0];
      =     L 1.6;
      BLD   103;
      A     DIX [AR2,P#116.2];
      =     L 1.7;
      BLD   103;
      CALL  "HF3_B_T_W_FC51" (
           Bit_0                    := L 0.0,
           Bit_1                    := L 0.1,
           Bit_2                    := L 0.2,
           Bit_3                    := L 0.3,
           Bit_4                    := L 0.4,
           Bit_5                    := L 0.5,
           Bit_6                    := L 0.6,
           Bit_7                    := L 0.7,
           Bit_8                    := L 1.0,
           Bit_9                    := L 1.1,
           Bit_10                   := L 1.2,
           Bit_11                   := L 1.3,
           Bit_12                   := L 1.4,
           Bit_13                   := L 1.5,
           Bit_14                   := L 1.6,
           Bit_15                   := L 1.7,
           Word1                    := #ToHMI);
      NOP   0;
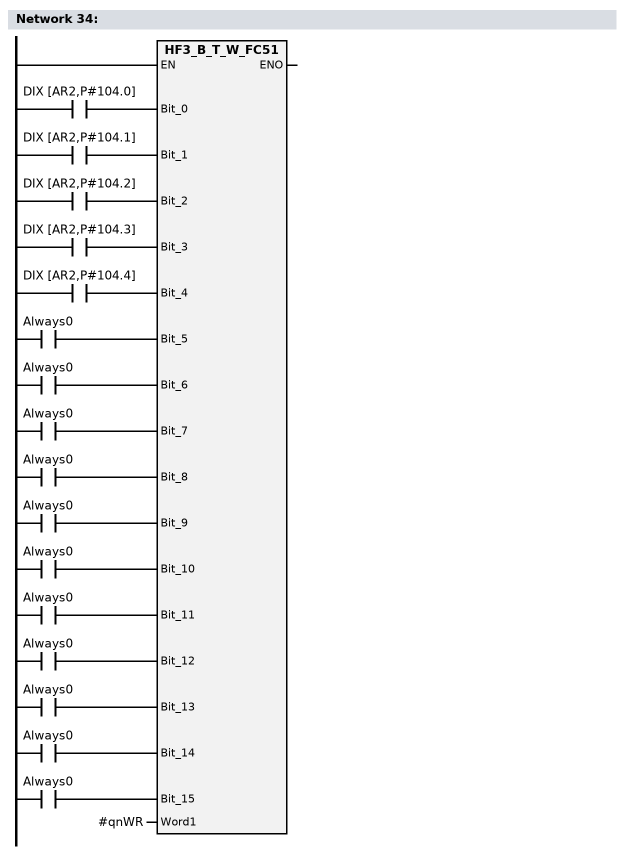
NETWORK
TITLE =
      A     DIX [AR2,P#104.0];
      =     L 0.0;
      BLD   103;
      A     DIX [AR2,P#104.1];
      =     L 0.1;
      BLD   103;
      A     DIX [AR2,P#104.2];
      =     L 0.2;
      BLD   103;
      A     DIX [AR2,P#104.3];
      =     L 0.3;
      BLD   103;
      A     DIX [AR2,P#104.4];
      =     L 0.4;
      BLD   103;
      A     "Always0";
      =     L 0.5;
      BLD   103;
      A     "Always0";
      =     L 0.6;
      BLD   103;
      A     "Always0";
      =     L 0.7;
      BLD   103;
      A     "Always0";
      =     L 1.0;
      BLD   103;
      A     "Always0";
      =     L 1.1;
      BLD   103;
      A     "Always0";
      =     L 1.2;
      BLD   103;
      A     "Always0";
      =     L 1.3;
      BLD   103;
      A     "Always0";
      =     L 1.4;
      BLD   103;
      A     "Always0";
      =     L 1.5;
      BLD   103;
      A     "Always0";
      =     L 1.6;
      BLD   103;
      A     "Always0";
      =     L 1.7;
      BLD   103;
      CALL  "HF3_B_T_W_FC51" (
           Bit_0                    := L 0.0,
           Bit_1                    := L 0.1,
           Bit_2                    := L 0.2,
           Bit_3                    := L 0.3,
           Bit_4                    := L 0.4,
           Bit_5                    := L 0.5,
           Bit_6                    := L 0.6,
           Bit_7                    := L 0.7,
           Bit_8                    := L 1.0,
           Bit_9                    := L 1.1,
           Bit_10                   := L 1.2,
           Bit_11                   := L 1.3,
           Bit_12                   := L 1.4,
           Bit_13                   := L 1.5,
           Bit_14                   := L 1.6,
           Bit_15                   := L 1.7,
           Word1                    := #qnWR);
      NOP   0;
END_FUNCTION_BLOCK

FUNCTION_BLOCK "HF3_VRV_FB2541"	// FB 2541
VERSION : 0.1
VAR
  VRV : FB 2542;
END_VAR
BEGIN
NETWORK
TITLE =
      BLD   14;
      =     L 7.0;
      L     DINO;
      T     LW 5;
      CDB;
      OPN   DI [LW 5];
      TAR2  LD 1;
      OPN   DI 6001;
      L     DIW 8;
      OPN   DI [LW 5];
      T     #VRV.SCtrl;
      +AR2  P#0.0;
      UC    "HF3_VRV_FB2542";
      LAR2  LD 1;
      CDB;
      BLD   15;
      NOP   0;
END_FUNCTION_BLOCK

FUNCTION_BLOCK "HF3_VRV_FB2542"	// FB 2542
VERSION : 0.1
VAR_INPUT
  SCtrl : WORD ;	//上位控制命令
  CommOK : BOOL ;	//通信状态
  Out_M1_Run : BOOL ;	//室外机一运行
  Out_M2_Run : BOOL ;	//室外机二运行
  Out_M3_Run : BOOL ;	//室外机三运行
  PT : TIME ;	//超时时间
END_VAR
VAR_OUTPUT
  qtWR : ARRAY  [0 .. 1 ] OF //0-全开1-全关
  BOOL ;
END_VAR
VAR
  Ton1 : SFB 4;
  Ton2 : SFB 4;
  SCtrl_Temp : ARRAY  [0 .. 15 ] OF //0-全开1-全关
  BOOL ;
  Ctrl : ARRAY  [0 .. 15 ] OF //0-全开1-全关
  BOOL ;
  Latch : ARRAY  [0 .. 15 ] OF //0-开锁定1-关锁定
  BOOL ;
  DO_Temp : ARRAY  [0 .. 15 ] OF //0-全开1-全关
  BOOL ;
  SingTout : BOOL ;
  QTout : BOOL ;
  Timeout : BOOL ;
  McFlag : BOOL ;	//检修牌
END_VAR
BEGIN
NETWORK
TITLE =
      BLD   1;
      =     L 4.0;
      TAR2  LD 0;
      L     #SCtrl;
      T     LW 5;
      L     DINO;
      T     LW 7;
      +AR2  P#54.0;
      TAR2;
      LAR2  LD 0;
      T     LD 9;
      UC    "HF3_W_T_B_FC54";
      {     P#L 5.0, P#L 7.0 };
      LAR2  LD 0;
      BLD   2;
      NOP   0;
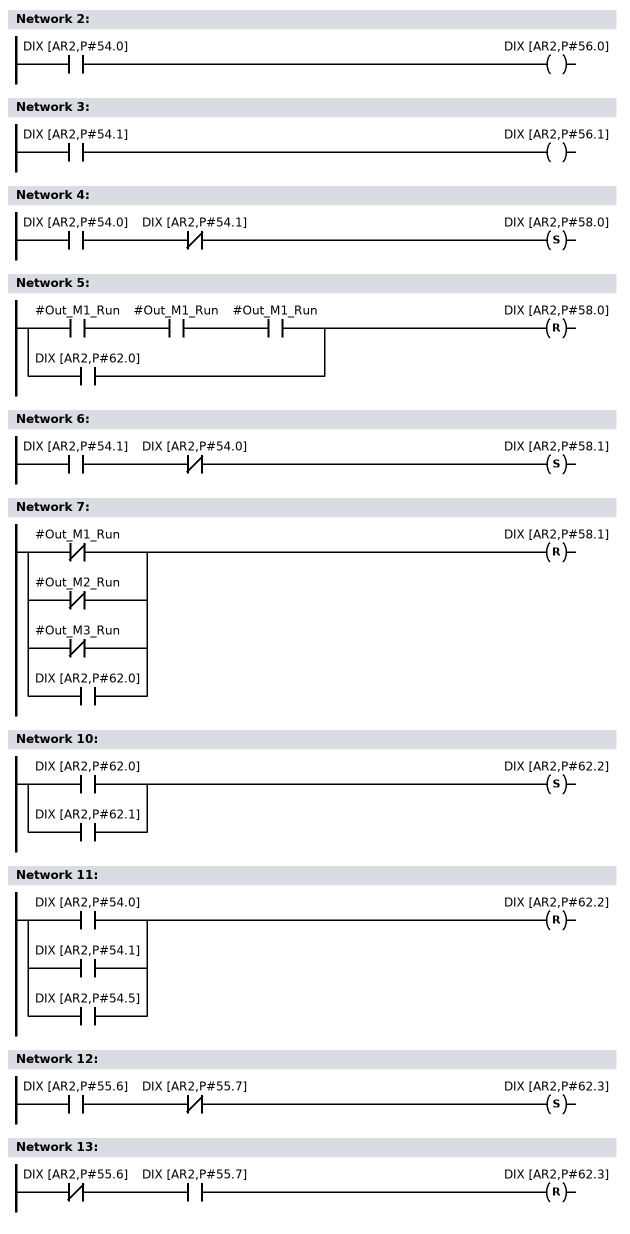
NETWORK
TITLE =
      A     DIX [AR2,P#54.0];
      =     DIX [AR2,P#56.0];
NETWORK
TITLE =
      A     DIX [AR2,P#54.1];
      =     DIX [AR2,P#56.1];
NETWORK
TITLE =
      A     DIX [AR2,P#54.0];
      AN    DIX [AR2,P#54.1];
      S     DIX [AR2,P#58.0];
NETWORK
TITLE =
      A     #Out_M1_Run;
      A     #Out_M1_Run;
      A     #Out_M1_Run;
      O     DIX [AR2,P#62.0];
      R     DIX [AR2,P#58.0];
NETWORK
TITLE =
      A     DIX [AR2,P#54.1];
      AN    DIX [AR2,P#54.0];
      S     DIX [AR2,P#58.1];
NETWORK
TITLE =
      ON    #Out_M1_Run;
      ON    #Out_M2_Run;
      ON    #Out_M3_Run;
      O     DIX [AR2,P#62.0];
      R     DIX [AR2,P#58.1];
NETWORK
TITLE =
      A(;
      O     DIX [AR2,P#58.0];
      O     DIX [AR2,P#58.1];
      );
      AN    DIX [AR2,P#54.0];
      AN    DIX [AR2,P#54.1];
      =     L 0.0;
      BLD   103;
      BLD   16;
      =     L 7.0;
      L     DINO;
      T     LW 5;
      CDB;
      OPN   DI [LW 5];
      TAR2  LD 1;
      A     L 0.0;
      =     DIX [AR2,P#10.0];
      L     DBD [AR2,P#4.0];
      T     DID [AR2,P#12.0];
      +AR2  P#10.0;
      UC    "TON";
      LAR2  LD 1;
      A     DIX [AR2,P#16.0];
      =     DBX [AR2,P#62.0];
      CDB;
      BLD   17;
      NOP   0;
NETWORK
TITLE =
      A(;
      O     DIX [AR2,P#60.0];
      O     DIX [AR2,P#60.1];
      );
      =     L 0.0;
      BLD   103;
      BLD   16;
      =     L 7.0;
      L     DINO;
      T     LW 5;
      CDB;
      OPN   DI [LW 5];
      TAR2  LD 1;
      A     L 0.0;
      =     DIX [AR2,P#32.0];
      L     DBD [AR2,P#4.0];
      T     DID [AR2,P#34.0];
      +AR2  P#32.0;
      UC    "TON";
      LAR2  LD 1;
      A     DIX [AR2,P#38.0];
      =     DBX [AR2,P#62.1];
      CDB;
      BLD   17;
      NOP   0;
NETWORK
TITLE =
      O     DIX [AR2,P#62.0];
      O     DIX [AR2,P#62.1];
      S     DIX [AR2,P#62.2];
NETWORK
TITLE =
      O     DIX [AR2,P#54.0];
      O     DIX [AR2,P#54.1];
      O     DIX [AR2,P#54.5];
      R     DIX [AR2,P#62.2];
NETWORK
TITLE =
      A     DIX [AR2,P#55.6];
      AN    DIX [AR2,P#55.7];
      S     DIX [AR2,P#62.3];
NETWORK
TITLE =
      AN    DIX [AR2,P#55.6];
      A     DIX [AR2,P#55.7];
      R     DIX [AR2,P#62.3];
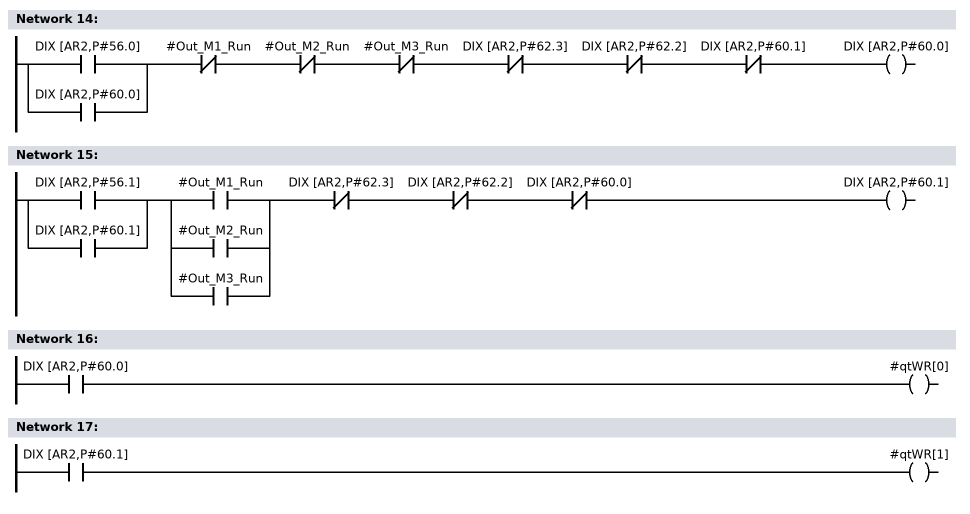
NETWORK
TITLE =
      A(;
      O     DIX [AR2,P#56.0];
      O     DIX [AR2,P#60.0];
      );
      AN    #Out_M1_Run;
      AN    #Out_M2_Run;
      AN    #Out_M3_Run;
      AN    DIX [AR2,P#62.3];
      AN    DIX [AR2,P#62.2];
      AN    DIX [AR2,P#60.1];
      =     DIX [AR2,P#60.0];
NETWORK
TITLE =
      A(;
      O     DIX [AR2,P#56.1];
      O     DIX [AR2,P#60.1];
      );
      A(;
      O     #Out_M1_Run;
      O     #Out_M2_Run;
      O     #Out_M3_Run;
      );
      AN    DIX [AR2,P#62.3];
      AN    DIX [AR2,P#62.2];
      AN    DIX [AR2,P#60.0];
      =     DIX [AR2,P#60.1];
NETWORK
TITLE =
      A     DIX [AR2,P#60.0];
      =     #qtWR[0];
NETWORK
TITLE =
      A     DIX [AR2,P#60.1];
      =     #qtWR[1];
END_FUNCTION_BLOCK

FUNCTION_BLOCK "HF3_SB_FB2551"	// FB 2551
VERSION : 0.1
VAR
  AT_A11 : FB 2552;
  PT_YSB : TIME ;
  AT_AYSB1 : FB 2552;
  AT_AYSB2 : FB 2552;
  AT_AYSB3 : FB 2552;
  AT_AYSB4 : FB 2552;
  AT_FSB : FB 2552;
  AT_QJFSB : FB 2552;
  AT_QJSB : FB 2552;
END_VAR
BEGIN
NETWORK
TITLE = AT_AYSB1
      A     "Always1";
      =     L 0.0;
      BLD   103;
      BLD   14;
      =     L 7.0;
      L     DINO;
      T     LW 5;
      CDB;
      OPN   DI [LW 5];
      TAR2  LD 1;
      L     2045;
      T     DIW [AR2,P#190.0];
      A     L 0.0;
      =     DIX [AR2,P#192.0];
      L     0;
      T     DIW [AR2,P#194.0];
      L     0;
      T     DIW [AR2,P#196.0];
      OPN   DI 6040;
      L     DIW 32;
      OPN   DI [LW 5];
      T     DIW [AR2,P#198.0];
      L     DBD [AR2,P#186.0];
      T     DID [AR2,P#200.0];
      OPN   DI 7005;
      L     DIW 312;
      OPN   DI [LW 5];
      T     DIW [AR2,P#204.0];
      +AR2  P#190.0;
      UC    "HF3_SB_FB2552";
      LAR2  LD 1;
      L     DIW [AR2,P#208.0];
      OPN   DI 6004;
      T     DIW 42;
      OPN   DI [LW 5];
      L     DIW [AR2,P#210.0];
      OPN   DI 6004;
      T     DIW 38;
      OPN   DI [LW 5];
      L     DIW [AR2,P#212.0];
      OPN   DI 6004;
      T     DIW 40;
      OPN   DI [LW 5];
      L     DID [AR2,P#214.0];
      OPN   DI 6004;
      T     DID 44;
      OPN   DI [LW 5];
      L     DIW [AR2,P#218.0];
      OPN   DI 6004;
      T     DIW 48;
      OPN   DI [LW 5];
      CDB;
      BLD   15;
      NOP   0;
NETWORK
TITLE = AT_AYSB2
      A     "Always1";
      =     L 0.0;
      BLD   103;
      BLD   14;
      =     L 7.0;
      L     DINO;
      T     LW 5;
      CDB;
      OPN   DI [LW 5];
      TAR2  LD 1;
      L     2045;
      T     DIW [AR2,P#376.0];
      A     L 0.0;
      =     DIX [AR2,P#378.0];
      L     12;
      T     DIW [AR2,P#380.0];
      L     12;
      T     DIW [AR2,P#382.0];
      OPN   DI 6040;
      L     DIW 34;
      OPN   DI [LW 5];
      T     DIW [AR2,P#384.0];
      L     DBD [AR2,P#186.0];
      T     DID [AR2,P#386.0];
      OPN   DI 7005;
      L     DIW 312;
      OPN   DI [LW 5];
      T     DIW [AR2,P#390.0];
      +AR2  P#376.0;
      UC    "HF3_SB_FB2552";
      LAR2  LD 1;
      L     DIW [AR2,P#394.0];
      OPN   DI 6004;
      T     DIW 54;
      OPN   DI [LW 5];
      L     DIW [AR2,P#396.0];
      OPN   DI 6004;
      T     DIW 50;
      OPN   DI [LW 5];
      L     DIW [AR2,P#398.0];
      OPN   DI 6004;
      T     DIW 52;
      OPN   DI [LW 5];
      L     DID [AR2,P#400.0];
      OPN   DI 6004;
      T     DID 56;
      OPN   DI [LW 5];
      L     DIW [AR2,P#404.0];
      OPN   DI 6004;
      T     DIW 60;
      OPN   DI [LW 5];
      CDB;
      BLD   15;
      NOP   0;
NETWORK
TITLE = AT_AYSB3
      A     "Always1";
      =     L 0.0;
      BLD   103;
      BLD   14;
      =     L 7.0;
      L     DINO;
      T     LW 5;
      CDB;
      OPN   DI [LW 5];
      TAR2  LD 1;
      L     2045;
      T     DIW [AR2,P#562.0];
      A     L 0.0;
      =     DIX [AR2,P#564.0];
      L     24;
      T     DIW [AR2,P#566.0];
      L     24;
      T     DIW [AR2,P#568.0];
      OPN   DI 6040;
      L     DIW 36;
      OPN   DI [LW 5];
      T     DIW [AR2,P#570.0];
      L     DBD [AR2,P#186.0];
      T     DID [AR2,P#572.0];
      OPN   DI 7005;
      L     DIW 312;
      OPN   DI [LW 5];
      T     DIW [AR2,P#576.0];
      +AR2  P#562.0;
      UC    "HF3_SB_FB2552";
      LAR2  LD 1;
      L     DIW [AR2,P#580.0];
      OPN   DI 6004;
      T     DIW 66;
      OPN   DI [LW 5];
      L     DIW [AR2,P#582.0];
      OPN   DI 6004;
      T     DIW 62;
      OPN   DI [LW 5];
      L     DIW [AR2,P#584.0];
      OPN   DI 6004;
      T     DIW 64;
      OPN   DI [LW 5];
      L     DID [AR2,P#586.0];
      OPN   DI 6004;
      T     DID 68;
      OPN   DI [LW 5];
      L     DIW [AR2,P#590.0];
      OPN   DI 6004;
      T     DIW 72;
      OPN   DI [LW 5];
      CDB;
      BLD   15;
      NOP   0;
NETWORK
TITLE = AT_AYSB4
      A     "Always1";
      =     L 0.0;
      BLD   103;
      BLD   14;
      =     L 7.0;
      L     DINO;
      T     LW 5;
      CDB;
      OPN   DI [LW 5];
      TAR2  LD 1;
      L     2035;
      T     DIW [AR2,P#748.0];
      A     L 0.0;
      =     DIX [AR2,P#750.0];
      L     0;
      T     DIW [AR2,P#752.0];
      L     0;
      T     DIW [AR2,P#754.0];
      OPN   DI 6040;
      L     DIW 38;
      OPN   DI [LW 5];
      T     DIW [AR2,P#756.0];
      L     DBD [AR2,P#186.0];
      T     DID [AR2,P#758.0];
      OPN   DI 7005;
      L     DIW 312;
      OPN   DI [LW 5];
      T     DIW [AR2,P#762.0];
      +AR2  P#748.0;
      UC    "HF3_SB_FB2552";
      LAR2  LD 1;
      L     DIW [AR2,P#766.0];
      OPN   DI 6004;
      T     DIW 78;
      OPN   DI [LW 5];
      L     DIW [AR2,P#768.0];
      OPN   DI 6004;
      T     DIW 74;
      OPN   DI [LW 5];
      L     DIW [AR2,P#770.0];
      OPN   DI 6004;
      T     DIW 76;
      OPN   DI [LW 5];
      L     DID [AR2,P#772.0];
      OPN   DI 6004;
      T     DID 80;
      OPN   DI [LW 5];
      L     DIW [AR2,P#776.0];
      OPN   DI 6004;
      T     DIW 84;
      OPN   DI [LW 5];
      CDB;
      BLD   15;
      NOP   0;
NETWORK
TITLE = AT_QJFSB
      A     "Always1";
      =     L 0.0;
      BLD   103;
      BLD   14;
      =     L 7.0;
      L     DINO;
      T     LW 5;
      CDB;
      OPN   DI [LW 5];
      TAR2  LD 1;
      L     2115;
      T     DIW [AR2,P#1306.0];
      A     L 0.0;
      =     DIX [AR2,P#1308.0];
      L     0;
      T     DIW [AR2,P#1310.0];
      L     0;
      T     DIW [AR2,P#1312.0];
      OPN   DI 6040;
      L     DIW 38;
      OPN   DI [LW 5];
      T     DIW [AR2,P#1314.0];
      L     DBD [AR2,P#186.0];
      T     DID [AR2,P#1316.0];
      OPN   DI 7005;
      L     DIW 312;
      OPN   DI [LW 5];
      T     DIW [AR2,P#1320.0];
      +AR2  P#1306.0;
      UC    "HF3_SB_FB2552";
      LAR2  LD 1;
      L     DIW [AR2,P#1324.0];
      OPN   DI 6004;
      T     DIW 102;
      OPN   DI [LW 5];
      L     DIW [AR2,P#1326.0];
      OPN   DI 6004;
      T     DIW 98;
      OPN   DI [LW 5];
      L     DIW [AR2,P#1328.0];
      OPN   DI 6004;
      T     DIW 100;
      OPN   DI [LW 5];
      L     DID [AR2,P#1330.0];
      OPN   DI 6004;
      T     DID 104;
      OPN   DI [LW 5];
      L     DIW [AR2,P#1334.0];
      OPN   DI 6004;
      T     DIW 108;
      OPN   DI [LW 5];
      CDB;
      BLD   15;
      NOP   0;
NETWORK
TITLE = AT_FSB
      A     "Always1";
      =     L 0.0;
      BLD   103;
      BLD   14;
      =     L 7.0;
      L     DINO;
      T     LW 5;
      CDB;
      OPN   DI [LW 5];
      TAR2  LD 1;
      L     2065;
      T     DIW [AR2,P#934.0];
      A     L 0.0;
      =     DIX [AR2,P#936.0];
      L     0;
      T     DIW [AR2,P#938.0];
      L     0;
      T     DIW [AR2,P#940.0];
      OPN   DI 6040;
      L     DIW 38;
      OPN   DI [LW 5];
      T     DIW [AR2,P#942.0];
      L     DBD [AR2,P#186.0];
      T     DID [AR2,P#944.0];
      OPN   DI 7005;
      L     DIW 312;
      OPN   DI [LW 5];
      T     DIW [AR2,P#948.0];
      +AR2  P#934.0;
      UC    "HF3_SB_FB2552";
      LAR2  LD 1;
      L     DIW [AR2,P#952.0];
      OPN   DI 6004;
      T     DIW 114;
      OPN   DI [LW 5];
      L     DIW [AR2,P#954.0];
      OPN   DI 6004;
      T     DIW 110;
      OPN   DI [LW 5];
      L     DIW [AR2,P#956.0];
      OPN   DI 6004;
      T     DIW 112;
      OPN   DI [LW 5];
      L     DID [AR2,P#958.0];
      OPN   DI 6004;
      T     DID 116;
      OPN   DI [LW 5];
      L     DIW [AR2,P#962.0];
      OPN   DI 6004;
      T     DIW 120;
      OPN   DI [LW 5];
      CDB;
      BLD   15;
      NOP   0;
END_FUNCTION_BLOCK

FUNCTION_BLOCK "HF3_SB_FB2552"	// FB 2552
//不要修改STL程序 不要改变IN OUT STAT 引脚参数在接口里的顺序
VERSION : 0.1
VAR_INPUT
  DB_NO : INT ;	//读DB号
  Multi : BOOL ;	//是否有多个水泵并线
  in_stradr : INT ;	//读命令状态开始地址
  out_stradr : INT ;	//slave_id开始地址
  SCtrl : WORD ;	//上位控制命令
  PT : TIME ;	//超时时间
  H_P_ALL_Ctrl : WORD ;	//全局控制命令
  FireAlarm : BOOL ;
END_VAR
VAR_OUTPUT
  Level_Value : INT ;	//水位mm
  ToHMI1 : WORD ;	//反馈上位信息1
  ToHMI2 : WORD ;	//反馈上位信息2
  RT : REAL ;	//泵运行时间
  SumFlt : INT ;	//泵故障次数
  SumRun : INT ;	//泵运行次数
END_VAR
VAR
  Ton1 : SFB 4;
  Ton2 : SFB 4;
  Ton3 : SFB 4;
  Ton4 : SFB 4;
  Ton5 : SFB 4;
  SingTout1 : BOOL ;	//一泵控制超时
  SingTout2 : BOOL ;	//二泵控制超时
  Timeout1 : BOOL ;	//一泵超时
  Timeout2 : BOOL ;	//二泵超时
  IN_RD1 : WORD ;
  IN_RD2 : WORD ;
  Comm_HB : WORD ;
  qnWR : WORD ;
  DI_Temp1 : ARRAY  [0 .. 15 ] OF //0自动1运行2运行
  BOOL ;
  DI_Temp2 : ARRAY  [0 .. 15 ] OF //水泵状态字
  BOOL ;
  DO_Temp : ARRAY  [0 .. 15 ] OF //01-1泵启停23-2泵启停 45-火灾信号
  BOOL ;
  Ctrl : ARRAY  [0 .. 15 ] OF //01-1泵启停23-2泵启停
  BOOL ;
  SCtrl_Temp : ARRAY  [0 .. 15 ] OF //01-1泵启停23-2泵启停
  BOOL ;
  Latch : ARRAY  [0 .. 7 ] OF //01-1泵启停锁定23-2泵启停锁定
  BOOL ;
  McFlag : BOOL ;	//挂检修牌
  QTout1 : BOOL ;	//一泵输出超时
  QTout2 : BOOL ;	//二泵输出超时
  H_P_ALL_Ctrl_Temp : ARRAY  [0 .. 15 ] OF BOOL ;
  CommOK_Temp : BOOL ;	//通信中间变量
  CommOK : BOOL ;	//通信正常
  RunFaultSun : FB 2006;
END_VAR
VAR_TEMP
  DI_reg : INT ;	//instance DB号
  db_no_temp : INT ;
  AR2_VALUE : DWORD ;	//AR2寄存器原始值
END_VAR
BEGIN
NETWORK
TITLE =
      A(;
      BLD   1;
      =     L 12.0;
      TAR2  LD 8;
      L     #SCtrl;
      T     LW 13;
      L     DINO;
      T     LW 15;
      +AR2  P#160.0;
      TAR2;
      LAR2  LD 8;
      T     LD 17;
      UC    "HF3_W_T_B_FC54";
      {     P#L 13.0, P#L 15.0 };
      LAR2  LD 8;
      BLD   2;
      A     BR;
      );
      JNB   _001;
      BLD   1;
      =     L 12.0;
      TAR2  LD 8;
      L     #H_P_ALL_Ctrl;
      T     LW 13;
      L     DINO;
      T     LW 15;
      +AR2  P#166.0;
      TAR2;
      LAR2  LD 8;
      T     LD 17;
      UC    "HF3_W_T_B_FC54";
      {     P#L 13.0, P#L 15.0 };
      LAR2  LD 8;
      BLD   2;
_001: NOP   0;
NETWORK
TITLE = 状态读取
//不要修改
      CLR;
      L     #DB_NO;
      T     #db_no_temp;
//当CP340接入多个水泵时
      L     P#0.0;
      LAR1;
      A     #Multi;	//1：多个水泵并线  0：单个泵
      JCN   sigl;
      L     #in_stradr;
      SLD   3;
      LAR1;
// AR1用于访问DB AR2用于访问DIB
//sigl：
// TAR2  
// T     #AR2_VALUE
// AD    DW#16#FFFFFF
// L     P##IN_RD1
// +D    
//  LAR2  
// 寄存器40002 、40003内容传递 通讯状态传递
sigl: OPN   DB [#db_no_temp];	//寄存器40002内容传递
      L     DBW [AR1,P#4.0];
// T     W [AR2,P#0.0]
      T     DIW [AR2,P#144.0];
      L     DBW [AR1,P#6.0];	//寄存器40003内容传递
// T     W [AR2,P#2.0]
      T     DIW [AR2,P#146.0];
      L     DBW [AR1,P#0.0];
// T     W [AR2,P#4.0]               //该设备通讯状态   0为正常
      T     DIW [AR2,P#148.0];
//水泵水位数值传递
//  L     #AR2_VALUE
//   AD    DW#16#FFFFFF
//    L     P##Level_Value
//    +D    
//   LAR2  
      L     DBW [AR1,P#8.0];
//T     W [AR2,P#0.0]               // 水泵水位赋值
      T     #Level_Value;
//恢复AR2中的初始值
//   L     #AR2_VALUE
//   LAR2  
NETWORK
TITLE =
      A(;
      BLD   1;
      =     L 12.0;
      TAR2  LD 8;
      L     DIW [AR2,P#144.0];
      T     LW 13;
      L     DINO;
      T     LW 15;
      +AR2  P#152.0;
      TAR2;
      LAR2  LD 8;
      T     LD 17;
      UC    "HF3_W_T_B_FC54";
      {     P#L 13.0, P#L 15.0 };
      LAR2  LD 8;
      BLD   2;
      A     BR;
      );
      JNB   _002;
      BLD   1;
      =     L 12.0;
      TAR2  LD 8;
      L     DIW [AR2,P#146.0];
      T     LW 13;
      L     DINO;
      T     LW 15;
      +AR2  P#154.0;
      TAR2;
      LAR2  LD 8;
      T     LD 17;
      UC    "HF3_W_T_B_FC54";
      {     P#L 13.0, P#L 15.0 };
      LAR2  LD 8;
      BLD   2;
_002: NOP   0;
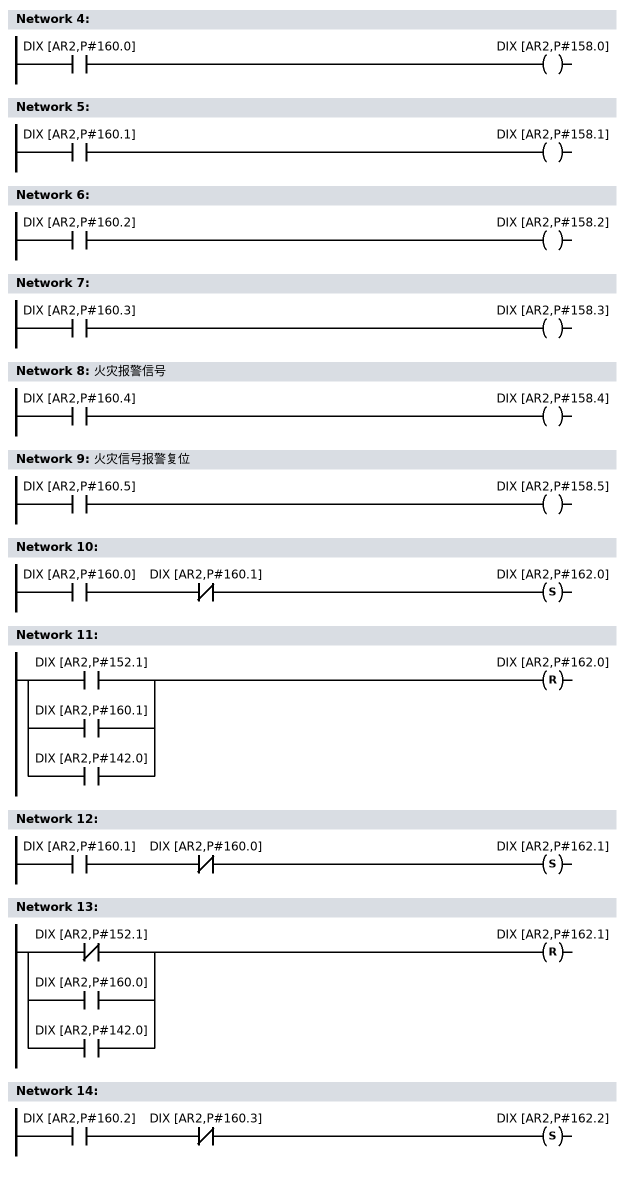
NETWORK
TITLE =
      A     DIX [AR2,P#160.0];
      =     DIX [AR2,P#158.0];
NETWORK
TITLE =
      A     DIX [AR2,P#160.1];
      =     DIX [AR2,P#158.1];
NETWORK
TITLE =
      A     DIX [AR2,P#160.2];
      =     DIX [AR2,P#158.2];
NETWORK
TITLE =
      A     DIX [AR2,P#160.3];
      =     DIX [AR2,P#158.3];
NETWORK
TITLE = 火灾报警信号
      A     DIX [AR2,P#160.4];
      =     DIX [AR2,P#158.4];
NETWORK
TITLE = 火灾信号报警复位
      A     DIX [AR2,P#160.5];
      =     DIX [AR2,P#158.5];
NETWORK
TITLE =
      A     DIX [AR2,P#160.0];
      AN    DIX [AR2,P#160.1];
      S     DIX [AR2,P#162.0];
NETWORK
TITLE =
      O     DIX [AR2,P#152.1];
      O     DIX [AR2,P#160.1];
      O     DIX [AR2,P#142.0];
      R     DIX [AR2,P#162.0];
NETWORK
TITLE =
      A     DIX [AR2,P#160.1];
      AN    DIX [AR2,P#160.0];
      S     DIX [AR2,P#162.1];
NETWORK
TITLE =
      ON    DIX [AR2,P#152.1];
      O     DIX [AR2,P#160.0];
      O     DIX [AR2,P#142.0];
      R     DIX [AR2,P#162.1];
NETWORK
TITLE =
      A     DIX [AR2,P#160.2];
      AN    DIX [AR2,P#160.3];
      S     DIX [AR2,P#162.2];
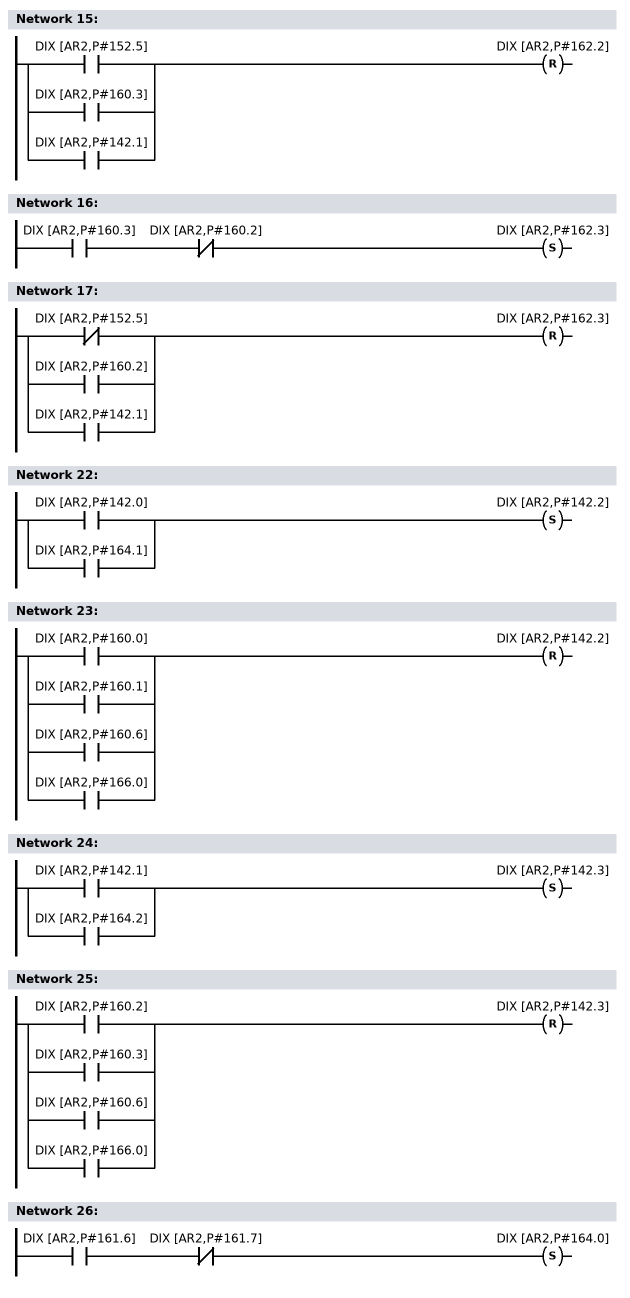
NETWORK
TITLE =
      O     DIX [AR2,P#152.5];
      O     DIX [AR2,P#160.3];
      O     DIX [AR2,P#142.1];
      R     DIX [AR2,P#162.2];
NETWORK
TITLE =
      A     DIX [AR2,P#160.3];
      AN    DIX [AR2,P#160.2];
      S     DIX [AR2,P#162.3];
NETWORK
TITLE =
      ON    DIX [AR2,P#152.5];
      O     DIX [AR2,P#160.2];
      O     DIX [AR2,P#142.1];
      R     DIX [AR2,P#162.3];
NETWORK
TITLE =
      A(;
      O     DIX [AR2,P#162.0];
      O     DIX [AR2,P#162.1];
      );
      AN    DIX [AR2,P#160.0];
      AN    DIX [AR2,P#160.1];
      =     L 8.0;
      BLD   103;
      BLD   16;
      =     L 15.0;
      L     DINO;
      T     LW 13;
      CDB;
      OPN   DI [LW 13];
      TAR2  LD 9;
      A     L 8.0;
      =     DIX [AR2,P#32.0];
      L     DBD [AR2,P#10.0];
      T     DID [AR2,P#34.0];
      +AR2  P#32.0;
      UC    "TON";
      LAR2  LD 9;
      A     DIX [AR2,P#38.0];
      =     DBX [AR2,P#142.0];
      CDB;
      BLD   17;
      NOP   0;
NETWORK
TITLE =
      A(;
      O     DIX [AR2,P#156.0];
      O     DIX [AR2,P#156.1];
      );
      =     L 8.0;
      BLD   103;
      BLD   16;
      =     L 15.0;
      L     DINO;
      T     LW 13;
      CDB;
      OPN   DI [LW 13];
      TAR2  LD 9;
      A     L 8.0;
      =     DIX [AR2,P#54.0];
      L     DBD [AR2,P#10.0];
      T     DID [AR2,P#56.0];
      +AR2  P#54.0;
      UC    "TON";
      LAR2  LD 9;
      A     DIX [AR2,P#60.0];
      =     DBX [AR2,P#164.1];
      CDB;
      BLD   17;
      NOP   0;
NETWORK
TITLE =
      A(;
      O     DIX [AR2,P#162.2];
      O     DIX [AR2,P#162.3];
      );
      AN    DIX [AR2,P#160.2];
      AN    DIX [AR2,P#160.3];
      =     L 8.0;
      BLD   103;
      BLD   16;
      =     L 15.0;
      L     DINO;
      T     LW 13;
      CDB;
      OPN   DI [LW 13];
      TAR2  LD 9;
      A     L 8.0;
      =     DIX [AR2,P#76.0];
      L     DBD [AR2,P#10.0];
      T     DID [AR2,P#78.0];
      +AR2  P#76.0;
      UC    "TON";
      LAR2  LD 9;
      A     DIX [AR2,P#82.0];
      =     DBX [AR2,P#142.1];
      CDB;
      BLD   17;
      NOP   0;
NETWORK
TITLE =
      A(;
      O     DIX [AR2,P#156.2];
      O     DIX [AR2,P#156.3];
      );
      =     L 8.0;
      BLD   103;
      BLD   16;
      =     L 15.0;
      L     DINO;
      T     LW 13;
      CDB;
      OPN   DI [LW 13];
      TAR2  LD 9;
      A     L 8.0;
      =     DIX [AR2,P#98.0];
      L     DBD [AR2,P#10.0];
      T     DID [AR2,P#100.0];
      +AR2  P#98.0;
      UC    "TON";
      LAR2  LD 9;
      A     DIX [AR2,P#104.0];
      =     DBX [AR2,P#164.2];
      CDB;
      BLD   17;
      NOP   0;
NETWORK
TITLE =
      O     DIX [AR2,P#142.0];
      O     DIX [AR2,P#164.1];
      S     DIX [AR2,P#142.2];
NETWORK
TITLE =
      O     DIX [AR2,P#160.0];
      O     DIX [AR2,P#160.1];
      O     DIX [AR2,P#160.6];
      O     DIX [AR2,P#166.0];
      R     DIX [AR2,P#142.2];
NETWORK
TITLE =
      O     DIX [AR2,P#142.1];
      O     DIX [AR2,P#164.2];
      S     DIX [AR2,P#142.3];
NETWORK
TITLE =
      O     DIX [AR2,P#160.2];
      O     DIX [AR2,P#160.3];
      O     DIX [AR2,P#160.6];
      O     DIX [AR2,P#166.0];
      R     DIX [AR2,P#142.3];
NETWORK
TITLE =
      A     DIX [AR2,P#161.6];
      AN    DIX [AR2,P#161.7];
      S     DIX [AR2,P#164.0];
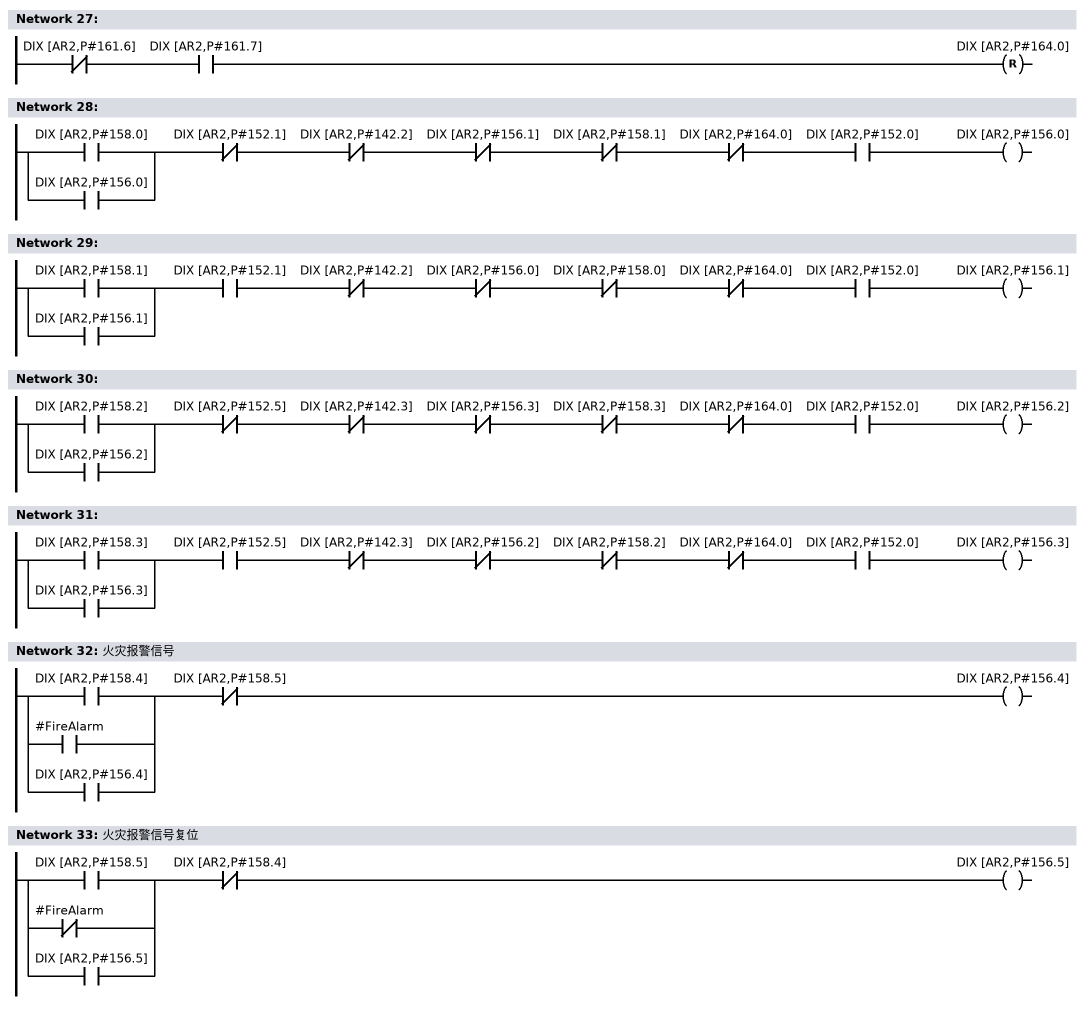
NETWORK
TITLE =
      AN    DIX [AR2,P#161.6];
      A     DIX [AR2,P#161.7];
      R     DIX [AR2,P#164.0];
NETWORK
TITLE =
      A(;
      O     DIX [AR2,P#158.0];
      O     DIX [AR2,P#156.0];
      );
      AN    DIX [AR2,P#152.1];
      AN    DIX [AR2,P#142.2];
      AN    DIX [AR2,P#156.1];
      AN    DIX [AR2,P#158.1];
      AN    DIX [AR2,P#164.0];
      A     DIX [AR2,P#152.0];
      =     DIX [AR2,P#156.0];
NETWORK
TITLE =
      A(;
      O     DIX [AR2,P#158.1];
      O     DIX [AR2,P#156.1];
      );
      A     DIX [AR2,P#152.1];
      AN    DIX [AR2,P#142.2];
      AN    DIX [AR2,P#156.0];
      AN    DIX [AR2,P#158.0];
      AN    DIX [AR2,P#164.0];
      A     DIX [AR2,P#152.0];
      =     DIX [AR2,P#156.1];
NETWORK
TITLE =
      A(;
      O     DIX [AR2,P#158.2];
      O     DIX [AR2,P#156.2];
      );
      AN    DIX [AR2,P#152.5];
      AN    DIX [AR2,P#142.3];
      AN    DIX [AR2,P#156.3];
      AN    DIX [AR2,P#158.3];
      AN    DIX [AR2,P#164.0];
      A     DIX [AR2,P#152.0];
      =     DIX [AR2,P#156.2];
NETWORK
TITLE =
      A(;
      O     DIX [AR2,P#158.3];
      O     DIX [AR2,P#156.3];
      );
      A     DIX [AR2,P#152.5];
      AN    DIX [AR2,P#142.3];
      AN    DIX [AR2,P#156.2];
      AN    DIX [AR2,P#158.2];
      AN    DIX [AR2,P#164.0];
      A     DIX [AR2,P#152.0];
      =     DIX [AR2,P#156.3];
NETWORK
TITLE = 火灾报警信号
      A(;
      O     DIX [AR2,P#158.4];
      O     #FireAlarm;
      O     DIX [AR2,P#156.4];
      );
      AN    DIX [AR2,P#158.5];
      =     DIX [AR2,P#156.4];
NETWORK
TITLE = 火灾报警信号复位
      A(;
      O     DIX [AR2,P#158.5];
      ON    #FireAlarm;
      O     DIX [AR2,P#156.5];
      );
      AN    DIX [AR2,P#158.4];
      =     DIX [AR2,P#156.5];
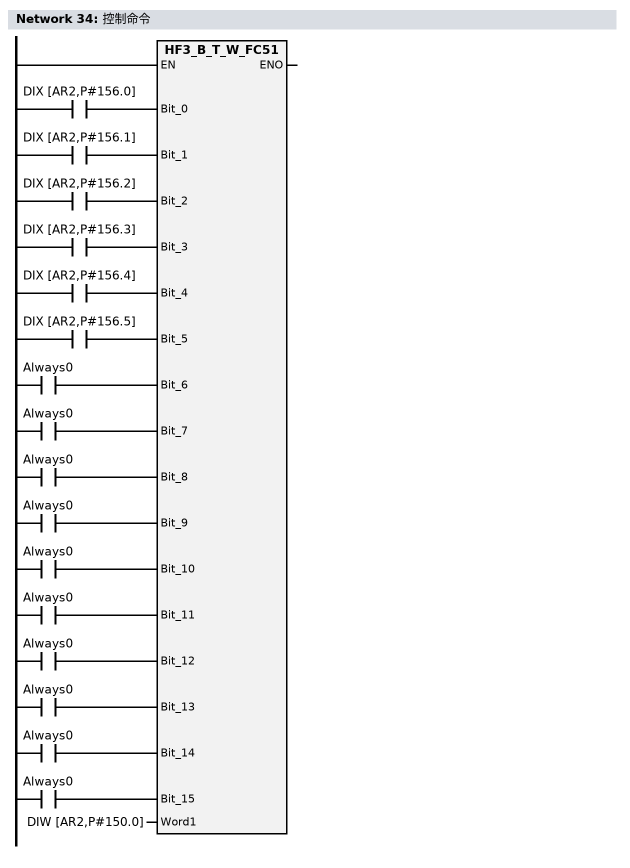
NETWORK
TITLE = 控制命令
      A     DIX [AR2,P#156.0];
      =     L 8.0;
      BLD   103;
      A     DIX [AR2,P#156.1];
      =     L 8.1;
      BLD   103;
      A     DIX [AR2,P#156.2];
      =     L 8.2;
      BLD   103;
      A     DIX [AR2,P#156.3];
      =     L 8.3;
      BLD   103;
      A     DIX [AR2,P#156.4];
      =     L 8.4;
      BLD   103;
      A     DIX [AR2,P#156.5];
      =     L 8.5;
      BLD   103;
      A     "Always0";
      =     L 8.6;
      BLD   103;
      A     "Always0";
      =     L 8.7;
      BLD   103;
      A     "Always0";
      =     L 9.0;
      BLD   103;
      A     "Always0";
      =     L 9.1;
      BLD   103;
      A     "Always0";
      =     L 9.2;
      BLD   103;
      A     "Always0";
      =     L 9.3;
      BLD   103;
      A     "Always0";
      =     L 9.4;
      BLD   103;
      A     "Always0";
      =     L 9.5;
      BLD   103;
      A     "Always0";
      =     L 9.6;
      BLD   103;
      A     "Always0";
      =     L 9.7;
      BLD   103;
      CALL  "HF3_B_T_W_FC51" (
           Bit_0                    := L 8.0,
           Bit_1                    := L 8.1,
           Bit_2                    := L 8.2,
           Bit_3                    := L 8.3,
           Bit_4                    := L 8.4,
           Bit_5                    := L 8.5,
           Bit_6                    := L 8.6,
           Bit_7                    := L 8.7,
           Bit_8                    := L 9.0,
           Bit_9                    := L 9.1,
           Bit_10                   := L 9.2,
           Bit_11                   := L 9.3,
           Bit_12                   := L 9.4,
           Bit_13                   := L 9.5,
           Bit_14                   := L 9.6,
           Bit_15                   := L 9.7,
           Word1                    := DIW [AR2,P#150.0]);
      NOP   0;
NETWORK
TITLE = 输出控制命令
//不要修改
      L     #out_stradr;
      SLD   3;
      LAR1;
      L     #db_no_temp;
      DEC   2;
      T     #db_no_temp;
//打开写共享数据块
      OPN   DB [#db_no_temp];
//控制命令给定
      CLR;
      L     #SCtrl;
      L     W#16#ABCD;
      <>I;
      JC    OFF;
//限制控制功能
      L     W#16#0;
      T     DIW [AR2,P#150.0];
OFF:  L     DIW [AR2,P#150.0];
      T     DBW [AR1,P#8.0];	//寄存器40005
NETWORK
TITLE = 通讯判断
      CLR;
      L     DIW [AR2,P#148.0];
      L     W#16#0;
      <>I;
      =     DIX [AR2,P#168.0];
      BLD   16;
      =     L 14.0;
      L     DINO;
      T     LW 12;
      CDB;
      OPN   DI [LW 12];
      TAR2  LD 8;
      A     DBX [AR2,P#168.0];
      =     DIX [AR2,P#120.0];
      L     L#3000;
      T     DID [AR2,P#122.0];
      +AR2  P#120.0;
      UC    "TON";
      LAR2  LD 8;
      A     DIX [AR2,P#126.0];
      =     DBX [AR2,P#168.1];
      CDB;
      BLD   17;
NETWORK
TITLE = 参数传递
      A     "Always0";
      =     L 8.0;
      BLD   103;
      A     DIX [AR2,P#152.5];
      =     L 8.1;
      BLD   103;
      A     DIX [AR2,P#152.6];
      =     L 8.2;
      BLD   103;
      A     DIX [AR2,P#152.7];
      =     L 8.3;
      BLD   103;
      A     DIX [AR2,P#153.0];
      =     L 8.4;
      BLD   103;
      A     DIX [AR2,P#153.7];
      =     L 8.5;
      BLD   103;
      A     "Always0";
      =     L 8.6;
      BLD   103;
      A     "Always0";
      =     L 8.7;
      BLD   103;
      A     "Always0";
      =     L 9.0;
      BLD   103;
      A     "Always0";
      =     L 9.1;
      BLD   103;
      A     "Always0";
      =     L 9.2;
      BLD   103;
      A     "Always0";
      =     L 9.3;
      BLD   103;
      A     "Always0";
      =     L 9.4;
      BLD   103;
      A     "Always0";
      =     L 9.5;
      BLD   103;
      A     "Always0";
      =     L 9.6;
      BLD   103;
      A     "Always0";
      =     L 9.7;
      BLD   103;
      A(;
      A     DIX [AR2,P#152.0];
      =     L 10.0;
      BLD   103;
      A     DIX [AR2,P#152.1];
      =     L 10.1;
      BLD   103;
      A     DIX [AR2,P#152.2];
      =     L 10.2;
      BLD   103;
      A     DIX [AR2,P#152.3];
      =     L 10.3;
      BLD   103;
      A     DIX [AR2,P#152.4];
      =     L 10.4;
      BLD   103;
      A     DIX [AR2,P#154.0];
      =     L 10.5;
      BLD   103;
      A     DIX [AR2,P#153.5];
      =     L 10.6;
      BLD   103;
      A     DIX [AR2,P#154.1];
      =     L 10.7;
      BLD   103;
      A     DIX [AR2,P#154.2];
      =     L 11.0;
      BLD   103;
      A     "Always0";
      =     L 11.1;
      BLD   103;
      A     "Always0";
      =     L 11.2;
      BLD   103;
      A     "Always0";
      =     L 11.3;
      BLD   103;
      A     DIX [AR2,P#142.2];
      =     L 11.4;
      BLD   103;
      A     DIX [AR2,P#142.3];
      =     L 11.5;
      BLD   103;
      A     DIX [AR2,P#164.0];
      =     L 11.6;
      BLD   103;
      AN    DIX [AR2,P#168.1];
      =     L 11.7;
      BLD   103;
      CALL  "HF3_B_T_W_FC51" (
           Bit_0                    := L 10.0,
           Bit_1                    := L 10.1,
           Bit_2                    := L 10.2,
           Bit_3                    := L 10.3,
           Bit_4                    := L 10.4,
           Bit_5                    := L 10.5,
           Bit_6                    := L 10.6,
           Bit_7                    := L 10.7,
           Bit_8                    := L 11.0,
           Bit_9                    := L 11.1,
           Bit_10                   := L 11.2,
           Bit_11                   := L 11.3,
           Bit_12                   := L 11.4,
           Bit_13                   := L 11.5,
           Bit_14                   := L 11.6,
           Bit_15                   := L 11.7,
           Word1                    := #ToHMI1);
      A     BR;
      );
      JNB   _003;
      CALL  "HF3_B_T_W_FC51" (
           Bit_0                    := L 8.0,
           Bit_1                    := L 8.1,
           Bit_2                    := L 8.2,
           Bit_3                    := L 8.3,
           Bit_4                    := L 8.4,
           Bit_5                    := L 8.5,
           Bit_6                    := L 8.6,
           Bit_7                    := L 8.7,
           Bit_8                    := L 9.0,
           Bit_9                    := L 9.1,
           Bit_10                   := L 9.2,
           Bit_11                   := L 9.3,
           Bit_12                   := L 9.4,
           Bit_13                   := L 9.5,
           Bit_14                   := L 9.6,
           Bit_15                   := L 9.7,
           Word1                    := #ToHMI2);
_003: NOP   0;
NETWORK
TITLE = 运行时间、故障次数
      A(;
      O     DIX [AR2,P#152.1];
      O     DIX [AR2,P#152.5];
      );
      =     L 8.0;
      BLD   103;
      A(;
      O     DIX [AR2,P#152.2];
      O     DIX [AR2,P#152.3];
      O     DIX [AR2,P#152.4];
      O     DIX [AR2,P#152.6];
      O     DIX [AR2,P#152.7];
      O     DIX [AR2,P#153.0];
      );
      =     L 8.1;
      BLD   103;
      A     M 20.3;
      =     L 8.2;
      BLD   103;
      A     DIX [AR2,P#161.4];
      =     L 8.4;
      BLD   103;
      A     DIX [AR2,P#161.5];
      =     L 8.5;
      BLD   103;
      BLD   14;
      =     L 15.0;
      L     DINO;
      T     LW 13;
      CDB;
      OPN   DI [LW 13];
      TAR2  LD 9;
      A     L 8.0;
      =     DIX [AR2,P#170.0];
      A     L 8.1;
      =     DIX [AR2,P#170.1];
      A     L 8.2;
      =     DIX [AR2,P#170.2];
      A     L 8.4;
      =     DIX [AR2,P#170.4];
      A     L 8.5;
      =     DIX [AR2,P#170.5];
      +AR2  P#170.0;
      UC    "HF3_RunFaultSum";
      LAR2  LD 9;
      L     DID [AR2,P#172.0];
      T     DBD [AR2,P#24.0];
      L     DIW [AR2,P#176.0];
      T     DBW [AR2,P#30.0];
      L     DIW [AR2,P#178.0];
      T     DBW [AR2,P#28.0];
      CDB;
      BLD   15;
      NOP   0;
END_FUNCTION_BLOCK

FUNCTION_BLOCK "HF3_3#SB_FB2561"	// FB 2561
VERSION : 0.1
VAR
  SB : FB 2562;
END_VAR
BEGIN
NETWORK
TITLE =
      BLD   14;
      =     L 6.0;
      L     DINO;
      T     LW 4;
      CDB;
      OPN   DI [LW 4];
      TAR2  LD 0;
      +AR2  P#0.0;
      UC    "HF3_3#SB_FB2562";
      LAR2  LD 0;
      CDB;
      BLD   15;
      NOP   0;
END_FUNCTION_BLOCK

